30: // 		udiIDXOFFS_MaxPos		: UDINT := 16#0000_000E;	// 8B
	fbADSWRITE.WRITE			:= TRUE;
	fbADSWRITE.IDXOFFS			:= 16#0000_000E;
	fbADSWRITE.LEN				:= 8;
	fbADSWRITE.SRCADDR			:= ADR(lrSetMaxPos);
	iStepWrite					:= iStepWrite + 5;
		
35: // 	End
	fbADSWRITE.WRITE			:= FALSE;
	IF NOT fbADSWRITE.BUSY AND NOT fbADSWRITE.ERR THEN
		bBusy 					:= FALSE;
		iStepWrite				:= 0;
	ELSIF fbADSWRITE.ERR THEN
		iStepWrite				:= 1000;
	END_IF
	
1000:
	bBusy 						:= FALSE;
	bError 						:= TRUE;
	udiErrorID					:= fbADSWRITE.ERRID;
	iStepWrite					:= 0;

END_CASE
END_ACTION

END_FUNCTION_BLOCK

// ---- POUs/NC/FB_CalculateSpeed.TcPOU
(********************************************************************************)
(*							Beckhoff Automation Poland							*)
(*							FB_CalculateSpeed  v1.0								*)
(*									28.8.2013									*)
(*			Blok funkcyjny obliczający predkosc z pozycji. z filtracją wyjscia	*)
(*						Wewnatrz wykorzystany blok FB_Filter					*)
(*______________________________________________________________________________*)
FUNCTION_BLOCK FB_CalculateSpeed
VAR_INPUT
	dwInput					: DWORD;     			(* zliczone impulsy z enkodera *)
	tSamplingTime 			: TIME;     			(* czas cyklu odczytu wejscia dwInput, musi byc rowony lub wiekszy od cyklu programu *)
	tT						: TIME;					(* stala czasowa filtracji - po tym czasie wyjscie przyjmuje ok 0,65 wartosci wejsciowej*)
END_VAR
VAR_OUTPUT
	rOut					: REAL; 				(* aktualna prędkość - unit/ms*)
	bError					: BOOL;					(* blad - czas probkowania mniejszy niz czas cyklu *)
END_VAR

VAR
	dwPrevInput				: DWORD;		 		(*liczba impulsów z poprzedniego odczytu*)
	rSamplingTime			: REAL; 				(*czas cyklu odczytu wejscia dwInput *)
	rDistance				: REAL;   				(*roznica w odczycie pomiedzy probkowaniami*)
	rRawOut					: REAL;   				(*prędkość przed filtracją*)
	dwBound					: DWORD;				(*granica wyznaczajaca przepetlenie*)
	BIndex					: BYTE;					(* nr tasku - do porowniania czasu cyklu *)
	tCycleTime				: TIME;					(* Ustawiony czas Tasku w ms*)
	tCurrentTime			: TIME;					(* aktualny czas *)
	tLastTime				: TIME;					(* poprzedni czas *)
	bCalculate				: BOOL;					(* sygnal do wykonania obliczen *)
	fbFilter 				: FB_Filter;			(* blok filtracji *)
	fbGETCURTASKINDEX		: GETCURTASKINDEX; 		(* Blok sprawdzajcy numer Tasku *)
END_VAR
VAR CONSTANT
	dwMaxInput				: DWORD := 4294967295;	(*maksymalna liczba impulsów*)
END_VAR

fbGETCURTASKINDEX(index=> BIndex);

dwBound 		:= dwMaxInput/4;								(*graniczna wartosc roznicy impulsow jest rowna 25% maksymalnej wartosci*)
tCycleTime		:= UDINT_TO_TIME(_TaskInfo[BIndex].CycleTime/10000);
bError			:= tSamplingTime < tCycleTime;					(* sprawdzenie warunku wykonalnosci *)
rSamplingTime	:= TIME_TO_REAL(tSamplingTime);
tCurrentTime 	:= TIME();										(* pobranie czasu plc *)
bCalculate 		:= (tCurrentTime - tLastTime) >= tSamplingTime; 	(* sprawdzamy czy nadszedl czas obliczen *)

IF bCalculate AND NOT bError  THEN
	IF dwInput < dwBound AND dwPrevInput > dwMaxInput- dwBound THEN 		(* Przepetlenie na + *)
		rDistance := DWORD_TO_REAL(dwInput - dwPrevInput);
	ELSIF dwInput > dwMaxInput- dwBound AND dwPrevInput < dwBound THEN 	(* Przepetlenie na - *)
		rDistance := DWORD_TO_REAL(dwInput - dwPrevInput);
	ELSE																		(* Bez przepetlenia zwykle odejmowanie *)
		rDistance := DWORD_TO_REAL(dwInput - dwPrevInput);
	END_IF
	rRawOut := rDistance/rSamplingTime;										(* Obliczenie predkosci *)
	(* Przepisanie starych wartosci *)
	tLastTime 		:= tCurrentTime;
	dwPrevInput 	:= dwInput;
END_IF

(*wygladzanie przebiegu*)
fbFIlter(In := rRawOut, tSamplingTime:= tSamplingTime, tMeasureTime:= tT, Out => rOut);

END_FUNCTION_BLOCK

// ---- POUs/Various/FB_Filter.TcPOU
(****************************************************************************************)
(*							Beckhoff Automation Poland									*)
(*								FB_Filter  v1											*)
(*									27.05.2008											*)
(*				Bloczek do filtru inercyjnego do wygladzania przebiegow					*)
(* 			Uwaga!! w nowych aplikacjach nalezy stosowac FB_FilterEx 					*)
(*______________________________________________________________________________________*)
FUNCTION_BLOCK FB_Filter
VAR_INPUT
	In:						REAL;(*sygnal wejsciowy*)
	tSamplingTime:			TIME;(*czas probkowania*)
	tMeasureTime:			TIME;(*stala czasowa*)
END_VAR
VAR_OUTPUT
	Out:					REAL;(*sygnal wyjsciowy*)
END_VAR
VAR
	czas_probkowania_real:	REAL;
	stala_czasowa_real:		REAL;
	CLOCK: 					TP;
	lastOut: 				REAL;
	lastStan: 				BOOL;
	stan: 					BOOL;
END_VAR

CLOCK();
clock.PT:=tSamplingTime;
czas_probkowania_real:=TIME_TO_REAL(tSamplingTime);
stala_czasowa_real:= TIME_TO_REAL(tMeasureTime);
IF CLOCK.Q=FALSE THEN
	CLOCK(IN:=FALSE);
	stan := NOT stan;
	CLOCK(IN:=TRUE);
END_IF
IF(lastStan <> stan) THEN
	Out:= lastOut + (In -lastOut)*czas_probkowania_real/stala_czasowa_real;
END_IF
lastOut:=Out;
lastStan:= stan;

END_FUNCTION_BLOCK

// ---- POUs/NC/FB_Enc20bitToDWORD.TcPOU
(********************************************************************************************)
(*							Beckhoff Automation Poland										*)
(*								FB_Enc20bitToDWORD  v2										*)
(*									20.07.2010												*)
(*	Blok funkcyjny do poszerzania zakresu odczytu z encoderow,								*)
(*	wartosc wejsciowa typu DWORD przystosowana do 20 bitow <0; 1048575>						*)
(*	przenoszona jest na wyjscie typu DWORD <0; 4294967295>									*)
(*	Przepetlenie wartosci wejsciowej nie powoduje w tym przypadku bledu						*)
(*__________________________________________________________________________________________*)
FUNCTION_BLOCK FB_Enc20bitToDWORD
VAR_INPUT
	dwInput: 		DWORD;					(* wartosc wejsciowa *)
END_VAR
VAR_IN_OUT
	dwOutput: 		DWORD;					(*wartosc wyjsciowa*)
END_VAR
VAR
	dwLastInput: 	DWORD;
	mask20: 		DWORD := 16#000FFFFF;	(*20 bitow, 1048575 Dec*)
	dwOutputHW:		DWORD; 					(*Gorna czesc dworda*)
	bFirstCycle:	BOOL := TRUE;
END_VAR
VAR CONSTANT
	dwLow: 			DWORD := 250000;
	dwHigh: 		DWORD := 800000;
END_VAR

dwInput := mask20 AND dwInput;

(*pierwszy cykl*)
IF bFirstCycle THEN
	dwOutputHW := dwOutput AND 16#FFF00000;
	bFirstCycle := FALSE;
ELSE
	IF dwInput < dwLow AND dwLastInput > dwHigh THEN
		(*Przekroczylismy zakres w gore*)
		dwOutputHW := dwOutputHW + 16#00100000;
	END_IF

	IF dwInput > dwHigh AND dwLastInput < dwLow THEN
		(*Przekroczylismy zakres w dol*)
		dwOutputHW := dwOutputHW - 16#00100000;
	END_IF
END_IF

dwLastInput := dwInput;
dwOutput := dwOutputHW + dwInput;

END_FUNCTION_BLOCK

// ---- POUs/NC/FB_EncIntToDint.TcPOU
(****************************************************************************************)
(*							Beckhoff Automation Poland									*)
(*								FB_EncIntToDint  v1.1									*)
(*									2.12.2010											*)
(*	Blok funkcyjny do poszerzania zakresu odczytu z encoderow,							*)
(*	wartosc wejsciowa typu UINT <-32768; 32767>											*)
(*	przenoszona jest na wyjscie typu UDINT <-2147483648; 2147483647>					*)
(*	Przepetlenie wartosci wejsciowej nie powoduje w tym przypadku bledu					*)
(*______________________________________________________________________________________*)
FUNCTION_BLOCK FB_EncIntToDint
VAR_INPUT
	iInput : 			INT; 		(* wartosc wejsciowa *)
	bReset : 			BOOL;
END_VAR
VAR
	iDelta: 			INT;
	iLastInput : 		INT;
END_VAR
VAR_IN_OUT
	diOutput: 			DINT;		(* wartosc wyjsciowa  - warto zrobic jako persistent*)
END_VAR

IF bReset THEN
	diOutput := 0;
ELSE
	iDelta := ( iInput - iLastInput);
	diOutput := diOutput + iDelta;
END_IF

iLastInput := iInput;

END_FUNCTION_BLOCK

// ---- POUs/NC/FB_EncWordtoDword.TcPOU
(****************************************************************************************************)
(*							Beckhoff Automation Poland												*)
(*								FB_EncWordToDword  v1.1												*)
(*									2.12.2010														*)
(*	Blok funkcyjny do poszerzania zakresu odczytu z encoderow,										*)
(*	wartosc wejsciowa typu WORD <0;  65535> przenoszona jest na wyjscie typu DWORD <0; 4294967295>	*)
(*	Przepetlenie wartosci wejsciowej nie powoduje w tym przypadku bledu								*)
(*__________________________________________________________________________________________________*)
FUNCTION_BLOCK FB_EncWordToDword
VAR_INPUT
	wInput: 		DWORD;		(* wartosc wejsciowa *)
	bReset: 		BOOL; 		(* reset wartosci *)
END_VAR
VAR_IN_OUT
	dwOutput: 		DWORD;		(*wartosc wyjsciowa - warto zrobic jako presistent *)
END_VAR
VAR
	wLastInput: 	DWORD;		(* Ostatnia wartosc *)
	dwOutputHW:		DWORD; 		(* Gorna czesc dworda*)
	bFirstCycle: 	BOOL := TRUE;
END_VAR
VAR CONSTANT
	wLow: 			DWORD := 15000;
	wHigh:			DWORD := 50000;
END_VAR

(*pierwszy cykl*)
IF bReset THEN
	dwOutput := 0;
	dwOutputHW := 0;
END_IF

IF bFirstCycle THEN
	dwOutputHW := dwOutput AND 16#FFFF0000; (* pobranie gornego worda *)
	bFirstCycle := FALSE;
ELSE
	IF wInput < wLow AND wLastInput > wHigh THEN
		(* Przekroczylismy zakres w gore *)
		dwOutputHW := dwOutputHW + 16#00010000;
	END_IF
	IF wInput > wHigh AND wLastInput < wLow THEN
		(*Przekroczylismy zakres w dol*)
		dwOutputHW := dwOutputHW - 16#00010000;
	END_IF
END_IF

wLastInput := wInput;
dwOutput := dwOutputHW + wInput;

END_FUNCTION_BLOCK

// ---- POUs/NC/FB_ForceLockUnlock.TcPOU
(************************************************************************************************)
(*							Beckhoff Automation Poland											*)
(*								FB_ForceLockUnlock  v1.0										*)
(*									2.12.2010													*)
(*	Blok funkcyjny pozwalający w prosty sposób włączać i wyłączac hamulec silnika AMxxxx 		*)
(*							Potrzebna biblioteka MC2Drive 										*)
(*______________________________________________________________________________________________*)
FUNCTION_BLOCK FB_ForceLockUnlock
VAR_INPUT
	bForceLock : 		BOOL;
	bForceUnlock: 		BOOL;
END_VAR
VAR_OUTPUT
	bError: 			BOOL;
	bUnlocked: 			BOOL;
END_VAR
VAR_IN_OUT
	Axis: 				AXIS_REF;
END_VAR
VAR
	wWriteData:			WORD; 				(*1 - lock, 2 - unlock *)
	wReadData: 			WORD;
	ftWrite: 			F_TRIG;
	Delay1: 			TOF;
	fbSoEWrite: 		FB_SoEWrite;
	fbSoERead: 			FB_SoERead;
	wWriteDataOld: 		WORD;
END_VAR

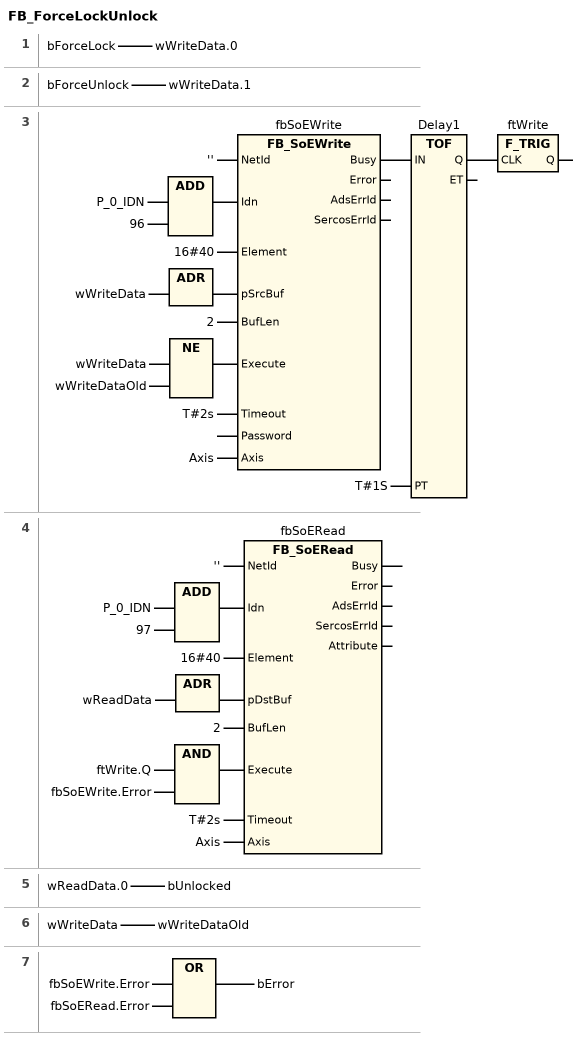
// NETWORK 1
wWriteData.0 := bForceLock;

// NETWORK 2
wWriteData.1 := bForceUnlock;

// NETWORK 3
fbSoEWrite(
    NetId := '',
    Idn := P_0_IDN + 96,
    Element := 16#40,
    pSrcBuf := ADR(wWriteData),
    BufLen := 2,
    Execute := wWriteData <> wWriteDataOld,
    Timeout := T#2s,
    Axis := Axis); // FB_SoEWrite
Delay1(IN := fbSoEWrite.Busy, PT := T#1S); // TOF
ftWrite(CLK := Delay1.Q); // F_TRIG

// NETWORK 4
fbSoERead(
    NetId := '',
    Idn := P_0_IDN + 97,
    Element := 16#40,
    pDstBuf := ADR(wReadData),
    BufLen := 2,
    Execute := ftWrite.Q AND fbSoEWrite.Error,
    Timeout := T#2s,
    Axis := Axis); // FB_SoERead

// NETWORK 5
bUnlocked := wReadData.0;

// NETWORK 6
wWriteDataOld := wWriteData;

// NETWORK 7
bError := fbSoEWrite.Error OR fbSoERead.Error;

END_FUNCTION_BLOCK

// ---- POUs/NC/FB_I2T_AX2000.TcPOU
(****************************************************************************)
(*							Beckhoff Automation Poland						*)
(*								FB_I2T_AX2000	 v1.0						*)
(*									27.05.2014								*)
(*							Blok odczytujący parametr I2T					*)
(* 							Wymaga biblioteki TcMc2Drive.lib 				*)
(*__________________________________________________________________________*)
FUNCTION_BLOCK FB_I2T_AX2000
VAR_INPUT
	bEnable					: BOOL := TRUE;
	sNetId					: T_AmsNetId; (* AMS Net ID of EtherCAT Master *)
	nSlaveAddr				: INT;
END_VAR
VAR_OUTPUT
	rI2T					: REAL;
	bBusy					: BOOL;
	bError					: BOOL;
	nErrId					: UDINT;
END_VAR
VAR
	fbEcCoESdoRead			: FB_EcCoESdoRead;
	tonWait200ms			: TON;
	dwI2T					: DWORD;
END_VAR

tonWait200ms(IN:= NOT tonWait200ms.Q AND bEnable, PT:=T#200MS );

fbEcCoESdoRead(
	sNetId:=sNetId ,
	nSlaveAddr:=INT_TO_UINT(nSlaveAddr),
	nSubIndex:=16#1 ,
	nIndex:=16#3559 ,
	pDstBuf:=ADR(dwI2T) ,
	cbBufLen:=SIZEOF(dwI2T) ,
	bExecute:=tonWait200ms.Q ,
	tTimeout:=t#2000ms ,
	bBusy=>bBusy ,
	bError=>bError ,
	nErrId=>nErrId );

rI2T := (DWORD_TO_REAL (dwI2T))/10.0;

END_FUNCTION_BLOCK

// ---- POUs/NC/FB_I2T_EL72x1.TcPOU
(************************************************************************************************)
(*							Beckhoff Automation Poland											*)
(*								FB_I2T_EL72x1	 v1.2											*)
(*							v1.1 - usuniecie /10, zmiana wyjść na typ USINT						*)
(*							v1.2 - poprawiony blad w nazwie zmiennej							*)
(*									24.10.2014													*)
(*							Blok odczytujący parametr I2T										*)
(* 							Wymaga biblioteki TcEtherCAT.lib 									*)
(*______________________________________________________________________________________________*)
FUNCTION_BLOCK FB_I2T_EL72x1
VAR_INPUT
(* A010:11 Amplifier I2T temperature  I2T model load Unit: % UINT8*)
(* A011:11 Motor I2T temperature  I2T model load Unit: % UINT8*)
	bEnable					: BOOL := TRUE; 		(* Pozwolenie na odczyt *)
	sNetId					: T_AmsNetId; 			(* AMS Net ID of EtherCAT Master *)
	nSlaveAddr				: UINT; 				(* Numer EtherCAT Slave *)
END_VAR
VAR_OUTPUT
	bBusy					: BOOL;
	bError					: BOOL;
	nErrorID				: UDINT;
	usiAmplifier_I2T		: USINT;
	usiMotor_I2T			: USINT;
END_VAR
VAR
(* Energy store/delete *)
	fbEcCoeSdoRead			: FB_EcCoESdoRead;
	bA010					: BOOL	:=TRUE;
	ftRead					: F_TRIG;
	tonWait200ms			: TON;
END_VAR

tonWait200ms(IN:=NOT tonWait200ms.Q AND bEnable, PT:=T#200MS );

fbEcCoeSdoRead.nIndex := SEL(bA010, 16#A011, 16#A010);
fbEcCoeSdoRead.pDstBuf := SEL(bA010, ADR(usiMotor_I2T), ADR(usiAmplifier_I2T));

fbEcCoeSdoRead(
	sNetId:= sNetId,
	nSlaveAddr:= nSlaveAddr,
	nSubIndex:= 16#11,
	cbBufLen:= 1,
	bExecute:= bEnable AND tonWait200ms.Q,
	bBusy=> bBusy,
	bError=> bError,
	nErrId=> nErrorID);

ftRead(CLK:= bBusy, Q=> );
bA010 := SEL(ftRead.Q, bA010, NOT bA010);

END_FUNCTION_BLOCK

// ---- POUs/NC/FB_PWM_BASIC.TcPOU
(********************************************************************************************************)
(*								Beckhoff Automation Poland												*)
(* 									FB_PWM_BASIC v1.1													*)
(* 										22.04.2010														*)
(*	v 1.1 - dodano bEnable, rCycleTime, początkowa faza to wyjście załączone, końcowa wyłączone			*)
(* 		Blok funkcyjny sterowania wyjsciem bOut typu BOOL na zasadzie modulowania szerokosci impulsu.	*)
(*					 Dokladnosc szerokosci impulsu  do 1 cylku sterownika.								*)
(* 							Konieczne jest dodanie biblioteki TcSystem									*)
(*______________________________________________________________________________________________________*)
FUNCTION_BLOCK FB_PWM_BASIC
VAR_INPUT
	bEnable: 			BOOL	:=TRUE;	(* Pozwolenie na działanie bloczka *)
	tPulseWidth: 		TIME; 			(*Szerokosc impulsu = 100% w ms typ zmiennej TIME*)
	fUpPercent: 		REAL; 			(*Aktualne procentowe wypelnienie impulsu*)
	rCycleTime: 		REAL;			(* Czas cylku - task, w milisekundach *)
END_VAR
VAR_OUTPUT
	bOut: 				BOOL;			(* Wyjscie *)
	wOn: 				WORD;			(* Liczba cykli z załączonym wyjściem *)
	wOff: 				WORD;			(* Liczba cykli z wyłaczonym wyjściem *)
END_VAR
VAR
	fCyclePulseWidth: 	REAL;  			(*Dlugosc impulsu = 100% w cyklach typ zmiennej REAL *)
	fCyclesOn: 			REAL;			(*Ilosc cykli, w ktorych sygnal jest zalaczony*)
	State: 				BYTE:=1;		(*Zmienna wyboru w instrukcji CASE*)
	(*Przeliczenie na pelne cykle*)
	wWidth: 			WORD;
	wCycleCounter:		WORD;			(*Licznik cykli zalaczenia/wylaczenia*)
	(*Przechowanie wartosci do porownania*)
	tPulseWidthOld: 	TIME	:= T#0MS;
	fUpPercentOld: 		REAL	:= -1;
END_VAR

IF bEnable THEN
	(*Przelicz tylko gdy zmienia sie dane*)
	IF tPulseWidth <> tPulseWidthOld OR fUpPercent <> fUpPercentOld THEN
		(*Sprawdzamy poprawnosc wprowadzonych danych*)
		IF fUpPercent <0 THEN fUpPercent := 0; END_IF
		IF fUpPercent > 100 THEN fUpPercent := 100; END_IF
		(*Obliczamy*)
		fCyclePulseWidth := TIME_TO_REAL(tPulseWidth)/rCycleTime; (*Dlugosc impulsu*)
		fCyclesOn := fCyclePulseWidth * fUpPercent/100;(*Cykle zalaczenia*)
	
		(*Przeliczamy na pelne cykle*)
		(*Opcja dla dokladniejszego przyblizenia impulsu On i Off*)
		wWidth := REAL_TO_WORD(fCyclePulseWidth);
		wOn := REAL_TO_WORD(fCyclesOn);
		(* Jeśli nie ma takiej potrzeby, nie wystawiaj wyjscia *)
		IF wOff = 0 THEN State := 0; END_IF
		wOff := REAL_TO_WORD(fCyclePulseWidth - fCyclesOn);
		(*Podstawiamy*)
		tPulseWidthOld := tPulseWidth;
		fUpPercentOld := fUpPercent;
	END_IF

	(*Albo wystawiamy TRUE albo FALSE*)
	CASE State OF
		0:
			bOut := FALSE;									(*Ustaw bOut na FALSE*)
			wCycleCounter := wCycleCounter  +  1;			(*Dodaj cykl do licznika*)
			IF wCycleCounter >= wOff THEN					(*Jezeli bylo bOut = FALSE wystarczajaca ilosc cykli to...*)
				wCycleCounter := 0;							(*Resetuj licznik*)
				IF wOff <> wWidth THEN State := 1; END_IF 	(*Przelacz tylko jesli ma byc kiedys bOut = TRUE*)
			END_IF
		1:
			bOut := TRUE;									(*Ustaw bOut na TRUE*)
			wCycleCounter := wCycleCounter  +  1;			(*Dodaj cykl do licznika*)
			IF wCycleCounter >= wOn THEN					(*Jezeli bylo bOut = TRUE wystarczajaca ilosc cykli to...*)
				wCycleCounter := 0;							(*Resetuj licznik*)
				IF wOn <> wWidth THEN State := 0; END_IF 	(*Przelacz tylko jesli ma byc kiedys bOut = FALSE*)
			END_IF
	END_CASE
ELSE
	bOut := FALSE;
	wCycleCounter := 0;
	State := 1;
END_IF

END_FUNCTION_BLOCK

// ---- POUs/NC/FB_SetBiasValue.TcPOU
(************************************************************************************************)
(*							Beckhoff Automation Poland											*)
(*								FB_SetBiasValue	 v1.0											*)
(*									12.04.2015													*)
(*							Blok wpisujący offset pozycji										*)
(* 							Wymaga biblioteki TcMc2.lib 										*)
(*______________________________________________________________________________________________*)
FUNCTION_BLOCK FB_SetBiasValue
VAR_INPUT
	bExecute			: BOOL; 		(* Narastajace zbocze aktywuje zapis *)
	sNetId				: T_AmsNetId;
	lrBias				: LREAL;
END_VAR
VAR_OUTPUT
	bBusy				: BOOL;
	bError				: BOOL;
	udiErrorID			: UDINT;
END_VAR
VAR_IN_OUT
	Axis				: AXIS_REF;
END_VAR
VAR
	fbADSWRITE			: ADSWRITE;
END_VAR

fbADSWRITE(
	NETID:= sNetId,
	PORT:= AMSPORT_R0_NC,
	IDXGRP:= 16#5000+Axis.NcToPlc.AxisId,
	IDXOFFS:= 7,
	LEN:= SIZEOF(lrBias),
	SRCADDR:= ADR(lrBias),
	WRITE:= bExecute,
	TMOUT:= ,
	BUSY=> bBusy,
	ERR=> bError,
	ERRID=> udiErrorID);

END_FUNCTION_BLOCK

// ---- POUs/NC/FB_TorqueMonitoringEL_Ex2.TcPOU
(****************************************************************************************************)
(*							Beckhoff Automation Poland												*)
(*							FB_TorqueMonitoringEL_Ex2 v1.1											*)
(*									25.11.2015														*)
(*																									*)
(*	Blok funkcyjny pozwala na monitorowanie i ograniczanie momentu oraz monitoring parametru I2T	*)
(*									dla EL7211.														*)
(*	Zmienne do zlinkowania zadeklarowane są wewnątrz bloku.		 									*)
(*	Ograniczenie i monitorowanie momentu															*)
(*	Ograniczenie momentu podawane jest przez wejście rTorqueLimit. 									*)
(*	Na wyjściu podana jest wartość surowa w %, jak i przeskalowana na A (prąd) i Nm (moment). 		*)
(*	Blok zwraca wartości bieżące, przefiltrowane i maksymalne. 										*)
(*	Wartości maksymalne mogą być wyzerowane za pomocą zmiennej bReset. 								*)
(*	Wewnętrznie wykorzystany jest blok FB_Filter.													*)
(*		I2T: 	Określamy okno czasowe pomiaru														*)
(* 	Wymaga biblioteki TcMc2Drive.lib 																*)
(*__________________________________________________________________________________________________*)
FUNCTION_BLOCK FB_TorqueMonitoringEL_Ex2
	VAR_INPUT
	bCalculate					: BOOL		:= TRUE;				(* Calculation request - initial value - TRUE *)
	bReset						: BOOL 		:= TRUE; 				(* Calculation request - initial value - TRUE *)
	rTorqueLimit				: REAL 		:= 100.0;			 	(* 0.0-100.0 %, rozdzielczość 0.1% *)
	tI2T_Window					: TIME;
END_VAR
VAR_OUTPUT
	bError						: BOOL; 							(* Communication error *)
	iErrorID					: INT;
	iTorque 			AT %I*	: INT; 								(* Raw data *)
	rCurrent					: REAL;								(* [A] *)
	rTorque						: REAL;								(* [Nm] *)
	rCurrentF					: REAL;								(* Filtered *)
	rTorqueF					: REAL;								(* Filtered *)
	rCurrentMax					: REAL;								(* Max *)
	rTorqueMax					: REAL;								(* Max *)
	rI2T						: REAL 		:= 0.0;
	rI2TMax						: REAL 		:= 0.0;
END_VAR
VAR_IN_OUT
	Axis						: AXIS_REF;
END_VAR
VAR
	iStep						: INT 		:= 0;

	rtCalculate					: R_TRIG;
	iTorqueLimitValue  	AT %Q*	:INT; 								(* Raw dara*)
	rFactor						: REAL;								(* iTorque -1000..1000 --> - rPeakCurrent .. rPeakCurrent *)
	rTorqueConstant				: REAL; 							(* [Nm/A] *)
	rPeakCurrent				: REAL; 							(* [A] *)
	rRatedCurrent				: REAL; 							(* [A] *)

	fbFilter					: FB_Filter;

	sNetId						: T_AmsNetId;
	uiSlaveAddr					: UINT;

	rI2T_pom					: REAL 		:= 0.0;
	rI2T_Window					: REAL;
	bFlag_1						: BOOL		:= FALSE;
	iCycles						: INT;
	rCycleTime_pom     	        : REAL;
	iCounter					: INT;
	rBuffer						: ARRAY[1..100] OF REAL;
	rBuffer_2					: ARRAY[1..100] OF REAL;

	fbMC_ReadDriveAddress		: MC_ReadDriveAddress;

	rCycleTime      		    : REAL;                             (* Ustawiony czas Tasku w ms*)
	fbGETCURTASKINDEX   		: GETCURTASKINDEX;                 	(* Blok sprawdzajcy numer Tasku *)
	BIndex                      : BYTE;                             (* Nr Tasku *)
(*-----------------------------------------------------------------------------------------------------------------------*)
	bRead						: BOOL;
	tTime						: TIME;
	wInfo						: WORD;
	dwPeakCurrent				: DWORD;
	dwStadnstillCurrent			: DWORD;
	dwRatedCurrent				: DWORD;
	dwTorqueConstant			: DWORD;
	dwDClinkCV					: DWORD		:= 0;
	fbEcCoESdoRead				: FB_EcCoESdoRead;
	BSubIndex					: BYTE;
	wIndex						: WORD;
	i							: INT		:= 1;
	pDstBuf						: POINTER TO DWORD;
	cbBufLen					: UDINT;
	ftRead						: F_TRIG;
	tonRead						: TON;
END_VAR

rtCalculate(CLK:= bCalculate, Q=> );
IF rtCalculate.Q THEN
	iStep := 0;
END_IF

CASE iStep OF

0:

(*Read drive adress*)

	bError:=FALSE;
	iErrorID:=0;
	fbMC_ReadDriveAddress(Execute := TRUE,Axis := Axis);
	iStep := iStep + 10;
10:
	fbMC_ReadDriveAddress(Axis := Axis);
	IF fbMC_ReadDriveAddress.Done THEN
		fbMC_ReadDriveAddress.Execute := FALSE;
		sNetId := fbMC_ReadDriveAddress.DriveAddress.NetID;
		uiSlaveAddr := fbMC_ReadDriveAddress.DriveAddress.SlaveAddress;
		iStep := iStep + 10;
	ELSIF fbMC_ReadDriveAddress.Error THEN
		iStep:=999;
		iErrorID:=UDINT_TO_INT(fbMC_ReadDriveAddress.ErrorID);
	END_IF
20:

(*Read cycle time*)

	fbGETCURTASKINDEX(index => BIndex);
	rCycleTime := UDINT_TO_REAL(_TaskInfo[BIndex].cycleTime)/10000.0;

(*Calculate algorithm sampling time*)

	rI2T_Window := TIME_TO_REAL(tI2T_Window);
	rCycleTime_pom := rI2T_Window/100 ;
	IF rCycleTime_pom < rCycleTime THEN
		rCycleTime_pom := rCycleTime;
	END_IF
	tTime := REAL_TO_TIME(rCycleTime_pom);
	iStep := iStep + 10;
30:

(*Chceck motor information using CoE*)

	bRead := TRUE;
	iStep := iStep + 10;
40:
	CoE_Read();
	IF NOT bRead THEN
		iStep := iStep + 10;
	END_IF
50:

(*Calculate current and torque value*)

	rCurrent := INT_TO_REAL(iTorque)*rPeakCurrent/1000;
	rTorque := rCurrent * rTorqueConstant;

(*Filter curent value*)

	fbFilter(In:= rCurrent, tSamplingTime:= REAL_TO_TIME(rCycleTime), tMeasureTime:= REAL_TO_TIME(rCycleTime_pom), Out=> rCurrentF);
	rTorqueF := rCurrentF * rTorqueConstant;

(*Save torque and current max values*)

	IF rCurrentMax < rCurrentF THEN
		rCurrentMax := rCurrentF;
		rTorqueMax := rTorqueF;
	END_IF

(*b_Flag_1 is set to TRUE when PLC cycle matches with algorythm sampling rate*)

	IF rCycleTime <> 0 THEN
		IF iCycles < rCycleTime_pom/rCycleTime  THEN
			iCycles := iCycles + 1;
			bFlag_1 := FALSE;
		ELSE
			iCycles := 0;
			bFlag_1 := TRUE;
		END_IF
	END_IF

(*Save momentary I2T values in ring buffer*)

	IF bFlag_1 THEN
		FOR iCounter:=1 TO 99 DO
			rBuffer[iCounter] := rBuffer[iCounter+1];
			rBuffer_2[iCounter] := rBuffer_2[iCounter+1];
		END_FOR
		rBuffer[100] := rCurrentF *rCurrentF* rCycleTime_pom;
		rBuffer_2[100] := rRatedCurrent *rRatedCurrent* rCycleTime_pom;
	END_IF
	rI2T := 0;
	rI2T_pom := 0;

(*Calculate I2T parameter*)

	FOR iCounter:=1 TO 100 DO
		rI2T := rI2T + rBuffer[iCounter];
		rI2T_pom := rI2T_pom + rBuffer_2[iCounter];
	END_FOR

(*Scale I2T to 0-100% range*)

	IF rI2T_pom <> 0  THEN
		rI2T := rI2T/rI2T_pom*100;
	END_IF

	IF rI2TMax < rI2T THEN
		rI2TMax := rI2T;
	END_IF

	IF bReset THEN
		rCurrentMax := 0;
		rTorqueMax := 0;
		rI2TMax := 0;
		FOR iCounter:=1 TO 100 DO
			rBuffer[iCounter] := 0;
			rBuffer_2[iCounter] := 0;
		END_FOR;
	END_IF
999:

(* Error occured *)

	bError:=TRUE;
	fbMC_ReadDriveAddress(Execute := FALSE,Axis := Axis);
	fbEcCoESdoRead(
	sNetId:= sNetId,
	nSlaveAddr:= uiSlaveAddr,
	nSubIndex:= BSubIndex,
	nIndex:= wIndex,
	pDstBuf:= pDstBuf,
	cbBufLen:= cbBufLen,
	bExecute := FALSE);

END_CASE;
iTorqueLimitValue := REAL_TO_INT(LIMIT(0.0,(rTorqueLimit)*10,1000.0));

ACTION CoE_Read:
CASE i OF
1:
	wIndex 			:= 16#6010;
	BSubIndex 		:= 1;
	pDstBuf 		:= ADR (wInfo);
	cbBufLen 		:= SIZEOF(wInfo);
2:
	wIndex 			:= 16#8011;
	BSubIndex 		:= 16#11;
	pDstBuf 		:= ADR (dwPeakCurrent);
	cbBufLen 		:= SIZEOF(dwPeakCurrent);
3:
	wIndex 			:= 16#8011;
	BSubIndex 		:= 16#12;
	pDstBuf 		:= ADR (dwRatedCurrent);
	cbBufLen 		:= SIZEOF(dwRatedCurrent);
4:
	wIndex 			:= 16#8011;
	BSubIndex 		:= 16#16;
	pDstBuf 			:= ADR (dwTorqueConstant);
	cbBufLen 		:= SIZEOF(dwTorqueConstant);
ELSE
	bRead 			:= FALSE;

	rRatedCurrent		:= DWORD_TO_REAL(dwRatedCurrent)/1000;
	rPeakCurrent 		:= DWORD_TO_REAL(dwPeakCurrent)/1000.0;
	rTorqueConstant	:= DWORD_TO_REAL(dwTorqueConstant)/1000.0;

	i := 1;
END_CASE

tonRead(IN := NOT tonRead.Q AND bRead, PT:= tTime, Q=> , ET=> );

fbEcCoESdoRead(
	sNetId:= sNetId,
	nSlaveAddr:= uiSlaveAddr,
	nSubIndex:= BSubIndex,
	nIndex:= wIndex,
	pDstBuf:= pDstBuf,
	cbBufLen:= cbBufLen,
	bExecute := tonRead.Q);
ftRead(CLK:= fbEcCoESdoRead.bBusy, Q=> );
IF ftRead.Q THEN
	IF fbEcCoESdoRead.bError THEN
		iErrorID := UDINT_TO_INT(fbEcCoESdoRead.nErrId);
		iStep:=999;
	END_IF
	i := i+1;
END_IF
END_ACTION

END_FUNCTION_BLOCK

// ---- POUs/NC/FB_TorqueMonitoringEx2.TcPOU
(****************************************************************************************************)
(*							Beckhoff Automation Poland												*)
(*							FB_TorqueMonitoringEx2 v1.1												*)
(*									23.04.2015														*)
(*			v1.1 - poprawiona obsługa błedów, optymalizacja obliczeń								*)
(*	Blok funkcyjny pozwala na monitorowanie i ograniczanie momentu oraz monitoring parametru I2T	*)
(*									dla AX5xxx.														*)
(*	Zmienne do zlinkowania zadeklarowane są wewnątrz bloku. 										*)
(*					Ograniczenie i monitorowanie momentu											*)
(*	Ograniczenie momentu podawane jest przez wejście rTorqueLimit. 									*)
(*	Na wyjściu podana jest wartość surowa w %, jak i przeskalowana na A (prąd) i Nm (moment).	 	*)
(*	Blok zwraca wartości bieżące, przefiltrowane i maksymalne. 										*)
(*	Wartości maksymalne mogą być wyzerowane za pomocą zmiennej bReset. 								*)
(*	Wewnętrznie wykorzystany jest blok FB_Filter.													*)
(*		I2T: 	Określamy okno czasowe pomiaru														*)
(* 	Wymaga biblioteki TcMc2Drive.lib 																*)
(*__________________________________________________________________________________________________*)
FUNCTION_BLOCK FB_TorqueMonitoringEx2
VAR_INPUT
	bCalculate					: BOOL		 := TRUE; 				(* Calculation request - initial value - TRUE *)
	bReset						: BOOL		 := TRUE;				(* Calculation request - initial value - TRUE *)
	rTorqueLimit				: REAL		 := 100.0; 				(* 0.0-100.0 %, rozdzielczość 0.1% *)
	tI2T_Window					: TIME		 :=T#1M;
END_VAR
VAR_OUTPUT
	bError						: BOOL; 							(* Communication error *)
	uiErrorID					: UINT;
	iTorque 			AT %I*	: INT; 								(* Raw data, linked to Torque feedback value AT, S-0-0084 *)
	rCurrent					: REAL; 							(* [A] *)
	rTorque						: REAL; 							(* [Nm] *)
	rCurrentF					: REAL;								(* Filtered *)
	rTorqueF					: REAL;								(* Filtered *)
	rCurrentMax					: REAL;								(* Max *)
	rTorqueMax					: REAL;								(* Max *)
	rI2T						: REAL; 							(* % nominal *)
	rI2TMax						: REAL;
END_VAR
VAR_IN_OUT
	Axis						: AXIS_REF;
END_VAR
VAR
	rtCalculate					: R_TRIG;
	fbSoERead					: FB_SoERead;
	iStep						: INT;
	P_0_0092_Value				: DWORD;
	P_0_0093_Value				: DWORD;
	P_0_0070_Value				: WORD;
	S_0_0111_Value				: DWORD;
	iBipolarTorqueLimitValue  	AT %Q*:		INT; 					(* Raw data, linked to Bipolar torque limit value MDT, S-0-0092 *)
	rPeakCurrent				: REAL; 							(* P_0_0092_Value in [A] *)
	rFactor						: REAL; 							(* iTorque -1000..1000 --> - rPeakCurrent .. rPeakCurrent *)
	rContinuousStallTorque		: REAL;								(* P_0_0070_Value [Nm] *)
	rContinuousStallCurrent		: REAL;								(* S_0_0111_Value [A] *)
	rTorqueConstant				: REAL; 							(* P_0_0070_Value/S_0_0111_Value [Nm/A] *)
	fbFilter					: FB_Filter;

	rI2T_pom					: REAL 		:= 0.0;
	rRatedCurrent				: REAL;	 							(* P_0_0093_Value in [A] *)
	rI2T_Window					: REAL;
	bFlag_1						: BOOL 		:= FALSE;
	bFlag_2						: BOOL 		:= FALSE;
	iCycles						: INT;
	iCycles_pom					: INT;
	rCycleTime_pom				: REAL;
	iCounter					: INT;
	rBuffer						: ARRAY[1..100] OF REAL;
	rBuffer_2					: ARRAY[1..100] OF REAL;

	rCycleTime					: REAL;                            	(* Ustawiony czas Tasku w ms*)
	fbGETCURTASKINDEX   		: GETCURTASKINDEX;                 	(* Blok sprawdzajcy numer Tasku *)
	BIndex						: BYTE;                             (* Nr Tasku *)
END_VAR

rtCalculate(CLK:= bCalculate, Q=> );
IF rtCalculate.Q THEN iStep := 0; END_IF

CASE iStep OF
	0: (*Init*)
	bError := FALSE;
	iStep := iStep+ 10;

	10: (*Read P_0_0092*)
	fbSoERead.Idn 		:= P_0_IDN + 92;
	fbSoERead.Element	:= EC_SOE_ELEMENT_VALUE;
	fbSoERead.pDstBuf	:= ADR(P_0_0092_Value);
	fbSoERead.BufLen	:= SIZEOF(P_0_0092_Value);
	fbSoERead.Execute	:= TRUE;
	iStep := iStep+ 5;

	15:
	IF NOT fbSoERead.Busy AND NOT fbSoERead.Error THEN
		rPeakCurrent := DWORD_TO_REAL(P_0_0092_Value)/1000.0;
		rFactor := DWORD_TO_REAL(P_0_0092_Value)/1000000.0;
		fbSoERead.Execute	:= FALSE;
		iStep := iStep+ 5;
	END_IF
	IF fbSoERead.Error THEN
		iStep := 100;
	END_IF

	20:
	(*Read P_0_0070*)
	fbSoERead.Idn 		:= P_0_IDN + 70;
	fbSoERead.Element	:= EC_SOE_ELEMENT_VALUE;
	fbSoERead.pDstBuf	:= ADR(P_0_0070_Value);
	fbSoERead.BufLen	:= SIZEOF(P_0_0070_Value);
	fbSoERead.Execute	:= TRUE;
	iStep := iStep+ 5;

	25:
	IF NOT fbSoERead.Busy AND NOT fbSoERead.Error THEN
		rContinuousStallTorque := WORD_TO_REAL(P_0_0070_Value)/100;
		fbSoERead.Execute	:= FALSE;
		iStep := iStep+ 5;
	END_IF
	IF fbSoERead.Error THEN
		iStep := 100;
	END_IF

	30: (* Read S_0_0111*)
	fbSoERead.Idn 		:= S_0_IDN + 111;
	fbSoERead.Element	:= EC_SOE_ELEMENT_VALUE;
	fbSoERead.pDstBuf	:= ADR(S_0_0111_Value);
	fbSoERead.BufLen	:= SIZEOF(S_0_0111_Value);
	fbSoERead.Execute	:= TRUE;
	iStep := iStep+ 5;

	35:
	IF NOT fbSoERead.Busy AND NOT fbSoERead.Error THEN
		rContinuousStallCurrent := DWORD_TO_REAL(S_0_0111_Value)/1000;
		rTorqueConstant := rContinuousStallTorque/rContinuousStallCurrent;
		fbSoERead.Execute	:= FALSE;
		iStep := iStep+ 5;
	END_IF
	IF fbSoERead.Error THEN
		iStep := 100;
	END_IF

	40: (* Read P_0_0093*)
	fbSoERead.Idn 		:= P_0_IDN + 93;
	fbSoERead.Element	:= EC_SOE_ELEMENT_VALUE;
	fbSoERead.pDstBuf	:= ADR(P_0_0093_Value);
	fbSoERead.BufLen	:= SIZEOF(P_0_0093_Value);
	fbSoERead.Execute	:= TRUE;
	iStep := iStep+ 5;

	45:
	IF NOT fbSoERead.Busy AND NOT fbSoERead.Error THEN
		rRatedCurrent := DWORD_TO_REAL(P_0_0093_Value)/1000;
		fbSoERead.Execute	:= FALSE;
		iStep := iStep+ 5;
	END_IF
	IF fbSoERead.Error THEN
		iStep := 100;
	END_IF

	50: (*Calculations*)
	rCurrent := INT_TO_REAL(iTorque) * rFactor;
	rTorque := rCurrent * rTorqueConstant;

	100:
	iStep := 0;
	fbSoERead(Execute:= FALSE,Axis:= Axis);
	bError := TRUE;
	uiErrorID := fbSoERead.AdsErrId;
END_CASE

(*Read cycle time*)
fbGETCURTASKINDEX(index => BIndex);
rCycleTime := UDINT_TO_REAL(_TaskInfo[BIndex].cycleTime)/10000.0;

(*Calculate algorithm sampling time*)
rI2T_Window := TIME_TO_REAL(tI2T_Window);
rCycleTime_pom := rI2T_Window/100 ;

IF rCycleTime_pom < rCycleTime THEN
	rCycleTime_pom := rCycleTime;
END_IF

(*Filter current value*)

fbFilter(In:= rCurrent, tSamplingTime:= REAL_TO_TIME(rCycleTime), tMeasureTime:= REAL_TO_TIME(rCycleTime_pom), Out=> rCurrentF);
rTorqueF := rCurrentF * rTorqueConstant;

(*Save torque and current max values*)
IF rCurrentMax < rCurrentF THEN
	rCurrentMax := rCurrentF;
	rTorqueMax := rTorqueF;
END_IF

(*b_Flag_1 is set to TRUE when PLC cycle matches with algorythm sampling rate*)

IF rCycleTime <> 0 THEN
	IF iCycles < rCycleTime_pom/rCycleTime  THEN
		iCycles := iCycles + 1;
		bFlag_1 := FALSE;
	ELSE
		iCycles := 0;
		bFlag_1 := TRUE;
	END_IF
END_IF

(*Save momentary I2T values in ring buffer*)

IF bFlag_1 THEN
	FOR iCounter :=1 TO 99 DO
		rBuffer[iCounter] := rBuffer[iCounter+1];
		rBuffer_2[iCounter] := rBuffer_2[iCounter+1];
	END_FOR
	rBuffer[100] := rCurrentF *rCurrentF* rCycleTime_pom;
	rBuffer_2[100] := rRatedCurrent *rRatedCurrent* rCycleTime_pom;
END_IF

rI2T := 0;
rI2T_pom := 0;

(*Calculate I2T parameter*)

FOR iCounter:=1 TO 100 BY 1 DO
	rI2T := rI2T + rBuffer[iCounter];
	rI2T_pom := rI2T_pom + rBuffer_2[iCounter];
END_FOR

(*Scale I2T to 0-100% range*)

IF rI2T_pom  <> 0  THEN
	rI2T := rI2T/rI2T_pom*100;
END_IF

IF rI2TMax < rI2T THEN
	rI2TMax := rI2T;
END_IF

IF bReset THEN
	rCurrentMax := 0;
	rTorqueMax := 0;
	rI2TMax := 0;
	FOR iCounter:=1 TO 100 BY 1 DO
		rBuffer[iCounter] := 0;
		rBuffer_2[iCounter] := 0;
	END_FOR;
END_IF
iBipolarTorqueLimitValue := REAL_TO_INT(LIMIT(0.0,(rTorqueLimit)*10,1000.0));

fbSoERead(
	NetId:= '',
	Timeout:= T#1s,
	Axis:= Axis);

END_FUNCTION_BLOCK

// ---- POUs/Switches/FB_2SwB.TcPOU
(****************************************************************************************)
(*							Beckhoff Automation Poland									*)
(*								FB_2SwB v1.1											*)
(*									9.11.2007											*)
(*				Blok funkcyjny symulujący pracę dwóch przycisków bistabilnych			*)
(*						 jako sterowania światłem schodowym								*)
(*______________________________________________________________________________________*)
FUNCTION_BLOCK FB_2SwB
VAR_INPUT
	bSwitch1:			BOOL;		(*Pierwszy przycisk bistabilny*)
	bSwitch2:			BOOL;		(*Drugi przycisk bistabilny*)
	bReset:				BOOL;		(*Przywrócenie stanu początkowego*)
END_VAR
VAR_OUTPUT
	bOut:				BOOL;		(*Wyjscie sterujące oświetleniem*)
END_VAR
VAR
	RTrig1:				R_TRIG;
	RTrig2:				R_TRIG;
	FTrig1:				F_TRIG;
	FTrig2:				F_TRIG;
END_VAR

RTrig1(CLK:= bSwitch1);
RTrig2(CLK:= bSwitch2);
FTrig1(CLK:= bSwitch1);
FTrig2(CLK:= bSwitch2);
bOut  := SEL(RTrig1.Q OR rTrig2.Q OR FTrig1.Q OR FTrig2.Q, bOut , NOT bOut );
IF bReset THEN bOut := FALSE; END_IF

END_FUNCTION_BLOCK

// ---- POUs/Switches/FB_2SwM.TcPOU
(****************************************************************************************)
(*							Beckhoff Automation Poland									*)
(*								FB_2SwM v1.1											*)
(*									9.11.2007											*)
(*				Blok funkcyjny symulujący pracę dwóch przycisków monostabilnych			*)
(*						 jako sterowania światłem schodowym								*)
(*______________________________________________________________________________________*)
FUNCTION_BLOCK FB_2SwM
VAR_INPUT
	bSwitch1:	BOOL;		(*Pierwszy przycisk monostabilny*)
	bSwitch2:	BOOL;		(*Drugi przycisk monostabilny*)
	bReset:		BOOL; 		(*Przywrócenie stanu początkowego*)
END_VAR
VAR_OUTPUT
	bOut:		BOOL; 		(*Wyjscie sterujące oświetleniem*)
END_VAR
VAR
	Trig1:		R_TRIG;
	Trig2:		R_TRIG;
END_VAR

Trig1(CLK:= bSwitch1);
Trig2(CLK:= bSwitch2);
bOut  := SEL(Trig1.Q OR Trig2.Q, bOut , NOT bOut );
IF bReset THEN bOut := FALSE; END_IF

END_FUNCTION_BLOCK

// ---- POUs/Switches/FB_Click.TcPOU
(********************************************************************************************************)
(*							Beckhoff Automation Poland													*)
(*								FB_Click	 v1.1														*)
(*								16.06.2008																*)
(*	Blok funkcyjny rozpoznajacy pojedyncze klikniecie, klikniecie podwojne lub nacisniecie przycisku	*)
(*______________________________________________________________________________________________________*)
FUNCTION_BLOCK FB_Click
VAR_INPUT
	bSwitch: 		BOOL;		 		(*Przycisk*)
	tTime: 			TIME 	:= T#1S; 	(*Czas kiedu mozna kliknac dwukrotnie*)
	tPress: 		TIME := T#500MS;	(*Rozpoznanie nacisniecia*)
END_VAR
VAR_OUTPUT
	bDouble: 		BOOL;(*Przyjmuje wartosc TRUE dla dwukrotnego klikniecia*)
	bSingle: 		BOOL;(*Przyjmuje wartosc TRUE dla pojedynczego klikniecia*)
	bPress: 		BOOL;(*Przyjmuje wartosc TRUE dla przytrzymania przycisku*)
END_VAR
VAR
	nCounter: 		SINT;
	timer: 			TON;
	timerPress: 	TON;
	rtrig: 			R_TRIG;
	ftrig: 			F_TRIG;
	pom: 			BOOL; 				(*zmienna pomocnicza*)
END_VAR

(*Zeby tylko przez jeden cykl byly ustawione wyjscia*)
bDouble := FALSE;
bSingle := FALSE;

timer(IN:= , PT:=tTime , Q=> , ET=> );
timerPress(IN:= bSwitch, PT:= tPress, Q=>bPress , ET=> );
rtrig(CLK:= bSwitch, Q=> );
ftrig(CLK:= bSwitch, Q=> );

(*Wyzerowanie licznika jak jest Press*)
IF timerPress.Q THEN
	nCounter := 0;
END_IF

(*Obsługa krótkiego sygnału*)
IF rtrig.Q THEN
	timer.IN := TRUE;
	pom := TRUE;
END_IF
IF ftrig.Q AND pom THEN
	pom := FALSE;
	nCounter := nCounter + 1;
END_IF

IF timer.Q THEN
	timer.IN := FALSE;
	IF nCounter = 1 THEN
		bSingle := TRUE;
	ELSIF nCounter > 1 THEN
		bDouble := TRUE;
	END_IF
	nCounter := 0;
END_IF

END_FUNCTION_BLOCK

// ---- POUs/Switches/FB_ClickCounterBit.TcPOU
(********************************************************************************************************)
(*							Beckhoff Automation Poland													*)
(*							FB_ClickCounterBit v1.0														*)
(*									18.02.2008															*)
(*				Blok funkcyjny zliczający ilość kliknięć i podający ją w formie bitu w bajcie			*)
(*______________________________________________________________________________________________________*)
FUNCTION_BLOCK FB_ClickCounterBit
VAR_INPUT
	bSwitch:		BOOL;(*Przycisk, którego kliknięcia zliczamy*)
	tInterval: 		TIME;(*max czas między kliknięciami*)
END_VAR
VAR_OUTPUT
	BOut:			BYTE;(*Zliczona ilość kliknięć*)
END_VAR
VAR
	Counting:		TOF;
	BAmount:		BYTE;
	RisingEdge:		R_TRIG;
	FallingEdge:	F_TRIG;
END_VAR

Counting(IN:=bSwitch , PT:= tInterval, Q=> , ET=> );
RisingEdge(CLK:= bSwitch, Q=> );
FallingEdge(CLK:= Counting.Q, Q=> );
IF RisingEdge.Q AND Counting.Q THEN
	BAmount := BAmount+1;
	BOut := 0;
END_IF
IF FallingEdge.Q THEN
	IF BAmount > 8 THEN
		BAmount := 8;
	END_IF(**)
	BOut := LREAL_TO_BYTE(EXPT(2,BAmount-1));
	BAmount := 0;
END_IF

END_FUNCTION_BLOCK

// ---- POUs/Switches/FB_ClickCounterByte.TcPOU
(********************************************************************************************)
(*							Beckhoff Automation Poland										*)
(*							FB_ClickCounterByte v1.0										*)
(*									18.02.2008												*)
(*				Blok funkcyjny zliczający ilość kliknięć i podający ją w formie bajtu		*)
(*__________________________________________________________________________________________*)
FUNCTION_BLOCK FB_ClickCounterByte
VAR_INPUT
	bSwitch:		BOOL;		(*Przycisk, którego kliknięcia zliczamy*)
	tInterval: 		TIME;		(*max czas między kliknięciami*)
END_VAR
VAR_OUTPUT
	BOut:			BYTE;		(*Zliczona ilość kliknięć*)
END_VAR
VAR
	Counting:		TOF;
	BAmount:		BYTE;
	RisingEdge:		R_TRIG;
	FallingEdge:	F_TRIG;
END_VAR

Counting(IN:=bSwitch , PT:= tInterval, Q=> , ET=> );
RisingEdge(CLK:= bSwitch, Q=> );
FallingEdge(CLK:= Counting.Q, Q=> );
IF RisingEdge.Q AND Counting.Q THEN
	BAmount := BAmount+1;
END_IF
IF FallingEdge.Q THEN
	BOut := BAmount;
	BAmount := 0;
ELSE
	BOut := 0;
END_IF

END_FUNCTION_BLOCK

// ---- POUs/Switches/FB_Dimmer1P.TcPOU
(****************************************************************************************)
(*							Beckhoff Automation Poland									*)
(*								FB_Dimmer1P v1.0										*)
(*									21.11.2007											*)
(*		Blok funkcyjny do przyciemniania/rozjaśniania za pomocą 1 przycisku bistabilnego*)
(*							wykorzystywany z KL2751										*)
(*______________________________________________________________________________________*)
FUNCTION_BLOCK FB_Dimmer1P
VAR_INPUT
	bSwitch:		BOOL;					(*Obsługiwany przycisk*)
	bReset:			BOOL; 					(*Reset bloku funkcyjnego przez funkcję centralną*)
END_VAR
VAR_OUTPUT
	iOut: 			INT;					(*Wyjscie - powinno byc zlinkowane z wyjściem modułu KL2751*)
END_VAR
VAR_IN_OUT
	iOldOut: 		INT;					(*Zapamiętanie stanu w yjścia*)
END_VAR
VAR
	tLong:			TIME	:=T#200MS;		(*Czas określający długie wciśnięcie przycisku*)
	iStep:			INT		:=100;			(*Krok zmany wyjścia*)
	Czas:			TON;
	Licznik:		CTU;
	iFunction:		INT;
	bLong: 			BOOL	:=TRUE;
	bShort: 		BOOL;
	ResetTrig:		R_TRIG;
END_VAR

(*Przywrócenie ustawień początkowych*)
ResetTrig(CLK:=bReset);
IF ResetTrig.Q THEN iFunction := 1; bLong := TRUE; bShort := FALSE;  END_IF;

(* Wykrycie dlugiego nacisniecia *)
Czas(IN:= bSwitch, PT:=tLong);
(* Rozpoznanie funkcji *)
Licznik(CU:= bSwitch, RESET:= Licznik.Q, PV:= 2);

IF Licznik.CV = 0 AND bSwitch THEN iFunction := 0; END_IF;(*wlaczany przycisk, byc moze rozjasnianie*)
IF Licznik.CV = 0 AND NOT bSwitch THEN iFunction := 1; END_IF;(*wylaczony przycisk, byc moze wlaczenie*)
IF Licznik.CV = 1 AND bSwitch THEN iFunction := 2; END_IF;(*wlaczany przycisk, byc moze sciemnianie*)
IF Licznik.CV = 1 AND NOT bSwitch THEN iFunction := 3; END_IF;(*wylaczony przycisk, byc moze wylaczenie*)
(*zapamietanie, ze bylo krotkie nacisniecie*)
IF bSwitch AND NOT Czas.Q THEN bLong := FALSE; END_IF;
IF NOT bSwitch AND NOT bLong THEN bShort := TRUE; END_IF;
(*zapamietanie, ze bylo dlugie nacisniecie*)
IF bSwitch AND Czas.Q THEN bLong := TRUE; bShort := FALSE; END_IF;

CASE iFunction OF

0:
(*przyciemnianie*)
IF bLong THEN
	iOut:=iOut-iStep;
	IF iOut<iStep THEN
		iOut :=0;
	END_IF
	iOldOut:=iOut;
END_IF;

1:
(*wylaczenie*)
IF bShort THEN iOut := 0; END_IF;

2:
(*rozjasnianie*)
IF bLong THEN
	iOut:=iOut+iStep;
	IF iOut<0THEN
		iOut :=32767;
	END_IF
	iOldOut:=iOut;
END_IF;

3:
(*wlaczenie*)
IF bShort THEN iOut:=iOldOut; END_IF;

END_CASE;

END_FUNCTION_BLOCK

// ---- POUs/Switches/FB_Dimmer1PMinMax.TcPOU
(****************************************************************************************)
(*							Beckhoff Automation Poland									*)
(*							FB_Dimmer1PMinMax v1.0										*)
(*									21.11.2007											*)
(*		Blok funkcyjny do przyciemniania/rozjaśniania za pomocą 1 przycisku bistabilnego*)
(*					z określaniem poziomu minimalnego i maksymalnego oświetlenia		*)
(*							wykorzystywany z KL2751										*)
(*______________________________________________________________________________________*)
FUNCTION_BLOCK FB_Dimmer1PMinMax
VAR_INPUT
	bSwitch:		BOOL;			(*Obsługiwany przycisk*)
	iMinLevel: 		INT; 			(*Minimalna wartość wyjścia*)
	iMaxLevel:	 	INT; 			(*Maksymalna wartość wyjścia*)
	bReset:			BOOL; 			(*Reset bloku funkcyjnego przez funkcję centralną*)
END_VAR
VAR_OUTPUT
	iOut: 			INT;			(*Wyjscie - powinno byc zlinkowane z wyjściem modułu KL2751*)
END_VAR
VAR_IN_OUT
	iOldOut: 		INT;			(*Zapamiętanie stanu w yjścia*)
END_VAR
VAR
	tLong:			TIME:=T#200MS;	(*Czas określający długie wciśnięcie przycisku*)
	iStep:			INT:=100;		(*Krok zmany wyjścia*)
	Czas:			TON;
	Licznik:		CTU;
	iFunction:		INT;
	bLong: 			BOOL:=TRUE;
	bShort: 		BOOL;
	ResetTrig:		R_TRIG;
END_VAR

(*Przywrócenie ustawień początkowych*)
ResetTrig(CLK:=bReset);
IF ResetTrig.Q THEN iFunction := 1; bLong := TRUE; bShort := FALSE;  END_IF;

(* Wykrycie dlugiego nacisniecia *)
Czas(IN:= bSwitch, PT:=tLong);
(* Rozpoznanie funkcji *)
Licznik(CU:= bSwitch, RESET:= Licznik.Q, PV:= 2);

IF Licznik.CV = 0 AND bSwitch THEN iFunction := 0; END_IF;(*wlaczany przycisk, byc moze rozjasnianie*)
IF Licznik.CV = 0 AND NOT bSwitch THEN iFunction := 1; END_IF;(*wylaczony przycisk, byc moze wlaczenie*)
IF Licznik.CV = 1 AND bSwitch THEN iFunction := 2; END_IF;(*wlaczany przycisk, byc moze sciemnianie*)
IF Licznik.CV = 1 AND NOT bSwitch THEN iFunction := 3; END_IF;(*wylaczony przycisk, byc moze wylaczenie*)
(*zapamietanie, ze bylo krotkie nacisniecie*)
IF bSwitch AND NOT Czas.Q THEN bLong := FALSE; END_IF;
IF NOT bSwitch AND NOT bLong THEN bShort := TRUE; END_IF;
(*zapamietanie, ze bylo dlugie nacisniecie*)
IF bSwitch AND Czas.Q THEN bLong := TRUE; bShort := FALSE; END_IF;

CASE iFunction OF

0:
(*przyciemnianie*)
IF bLong THEN
	iOut:=iOut-iStep;
	IF iOut<iMinLevel+iStep THEN
		iOut :=iMinLevel;
	END_IF
	iOldOut:=iOut;
END_IF;

1:
(*wylaczenie*)
IF bShort THEN iOut := 0; END_IF;

2:
(*rozjasnianie*)
IF bLong THEN
	iOut:=iOut+iStep;
	IF iOut<0 OR iOut>iMaxLevel THEN
		iOut :=iMaxLevel;
	END_IF
	iOldOut:=iOut;
END_IF;

3:
(*wlaczenie*)
IF bShort THEN iOut:=iOldOut; END_IF;

END_CASE;

END_FUNCTION_BLOCK

// ---- POUs/Switches/FB_Dimmer2P.TcPOU
(********************************************************************************************)
(*							Beckhoff Automation Poland										*)
(*								FB_Dimmer2P v1.0											*)
(*									21.11.2007												*)
(*		Blok funkcyjny do przyciemniania/rozjaśniania za pomocą 1 przycisków bistabilnych	*)
(*							wykorzystywany z KL2751											*)
(*__________________________________________________________________________________________*)
FUNCTION_BLOCK FB_Dimmer2P
VAR_INPUT
	bSwitchOnUp:			BOOL;			(*Przycisk 1*)
	bSwitchOffDown:			BOOL;			(*Przycisk 2*)
	bReset:					BOOL;			(*Reset bloku funkcyjnego przez funkcję centralną*)
END_VAR
VAR_OUTPUT
	iOut: 					INT;			(*Wyjscie - powinno byc zlinkowane z wyjściem modułu KL2751*)
END_VAR
VAR_IN_OUT
	iOldOut: 				INT;			(*Zapamiętanie stanu w yjścia*)
END_VAR
VAR
	iStep:					INT:=100;		(*Krok zmany wyjścia*)
	timeLong:		 		TIME:=T#200MS;	(*Czas długiego kliknięcia*)
	ftrig1:					F_TRIG;
	ftrig2:					F_TRIG;
	rtrig1:					R_TRIG;
	rtrig2:					R_TRIG;
	timer1:					TON;
	timer2:					TON;
	pom1: 					BOOL;
	bLong1: 				BOOL;
	bLong2: 				BOOL;
	pom2: 					BOOL;
	ResetTrig: 				R_TRIG;
END_VAR

(*Przywrócenie ustawień początkowych*)
ResetTrig(CLK:=bReset);
IF ResetTrig.Q THEN
	iOut :=0;
END_IF;
(*Wywołanie trigerow i timerow*)
timer1(PT:= timeLong);
ftrig1(CLK:= bSwitchOnUp);
rtrig1(CLK:= bSwitchOnUp);
timer2(PT:= timeLong);
ftrig2(CLK:= bSwitchOffDown);
rtrig2(CLK:= bSwitchOffDown);
(*Przycisk On i Up*)
(*Włączenie przycisku*)
IF rtrig1.Q THEN
	timer1.IN := TRUE;
	pom1 := TRUE;
	bLong1 := FALSE;
END_IF
(*Krótkie wciśnięcie*)
IF ftrig1.Q AND pom1 THEN
	pom1 := FALSE;
	timer1.IN := FALSE;
	iOut := iOldOut;
	bLong1 := FALSE;
END_IF
(*Długie wciśnięcie*)
IF timer1.Q THEN
	timer1.IN := FALSE;
	bLong1 := TRUE;
	pom1 := FALSE;
END_IF
(*Operacje gdy długi Up*)
IF bLong1 THEN
	iOut:=iOut+iStep;
	IF iOut<0THEN
		iOut :=32767;
	END_IF
	iOldOut:=iOut;
END_IF;
(*Wyłączenie długiego wciśnięcia*)
IF NOT bSwitchOnUp THEN
	bLong1 := FALSE;
END_IF

(*Przycisk Off i Down*)
(*Włączenie przycisku*)
IF rtrig2.Q THEN
	timer2.IN := TRUE;
	pom2 := TRUE;
	bLong2 := FALSE;
END_IF
(*Krótkie wciśnięcie*)
IF ftrig2.Q AND pom2 THEN
	pom2 := FALSE;
	timer2.IN := FALSE;
	iOut := 0;
	bLong2 := FALSE;
END_IF
(*Długie wciśnięcie*)
IF timer2.Q THEN
	timer2.IN := FALSE;
	bLong2 := TRUE;
	pom2 := FALSE;
END_IF
(*Operacje gdy długi Off*)
IF bLong2 THEN
	iOut:=iOut-iStep;
	IF iOut<iStep THEN
		iOut :=0;
	END_IF
	iOldOut:=iOut;
END_IF;
(*Wyłączenie długiego wciśnięcia*)
IF NOT bSwitchOffDown THEN
	bLong2 := FALSE;
END_IF

END_FUNCTION_BLOCK

// ---- POUs/Switches/FB_Dimmer2PMinMax.TcPOU
(********************************************************************************************)
(*							Beckhoff Automation Poland										*)
(*							FB_Dimmer2PMinMax v1.0											*)
(*									21.11.2007												*)
(*		Blok funkcyjny do przyciemniania/rozjaśniania za pomocą 1 przycisków bistabilnych	*)
(*					z określaniem poziomu minimalnego i maksymalnego oświetlenia			*)
(*							wykorzystywany z KL2751											*)
(*__________________________________________________________________________________________*)
FUNCTION_BLOCK FB_Dimmer2PMinMax
VAR_INPUT
	bSwitchOnUp:			BOOL;				(*Przycisk 1*)
	bSwitchOffDown:			BOOL;				(*Przycisk 2*)
	iMinLevel: 				INT; 				(*Minimalna wartość wyjścia*)
	iMaxLevel:		 		INT; 				(*Maksymalna wartość wyjścia*)
	bReset:					BOOL; 				(*Reset bloku funkcyjnego przez funkcję centralną*)
END_VAR
VAR_OUTPUT
	iOut: 					INT;				(*Wyjscie - powinno byc zlinkowane z wyjściem modułu KL2751*)
END_VAR
VAR_IN_OUT
	iOldOut: 				INT;				(*Zapamiętanie stanu w yjścia*)
END_VAR
VAR
	iStep:					INT:=100;			(*Krok zmany wyjścia*)
	timeLong:		 		TIME:=T#200MS;		(*Czas długiego kliknięcia*)
	ftrig1:					F_TRIG;
	ftrig2:					F_TRIG;
	rtrig1:					R_TRIG;
	rtrig2:					R_TRIG;
	timer1:					TON;
	timer2:					TON;
	pom1: 					BOOL;
	bLong1: 				BOOL;
	bLong2: 				BOOL;
	pom2: 					BOOL;
	ResetTrig: 				R_TRIG;
END_VAR

(*Przywrócenie ustawień początkowych*)
ResetTrig(CLK:=bReset);
IF ResetTrig.Q THEN
	iOut :=0;
END_IF;
(*Wywołanie trigerow i timerow*)
timer1(PT:= timeLong);
ftrig1(CLK:= bSwitchOnUp);
rtrig1(CLK:= bSwitchOnUp);
timer2(PT:= timeLong);
ftrig2(CLK:= bSwitchOffDown);
rtrig2(CLK:= bSwitchOffDown);
(*Przycisk On i Up*)
(*Włączenie przycisku*)
IF rtrig1.Q THEN
	timer1.IN := TRUE;
	pom1 := TRUE;
	bLong1 := FALSE;
END_IF
(*Krótkie wciśnięcie*)
IF ftrig1.Q AND pom1 THEN
	pom1 := FALSE;
	timer1.IN := FALSE;
	iOut := iOldOut;
	bLong1 := FALSE;
END_IF
(*Długie wciśnięcie*)
IF timer1.Q THEN
	timer1.IN := FALSE;
	bLong1 := TRUE;
	pom1 := FALSE;
END_IF
(*Operacje gdy długi Up*)
IF bLong1 THEN
	iOut:=iOut+iStep;
	IF iOut<0 OR iOut>iMaxLevel THEN
		iOut :=iMaxLevel;
	END_IF
	iOldOut:=iOut;
END_IF;
(*Wyłączenie długiego wciśnięcia*)
IF NOT bSwitchOnUp THEN
	bLong1 := FALSE;
END_IF

(*Przycisk Off i Down*)
(*Włączenie przycisku*)
IF rtrig2.Q THEN
	timer2.IN := TRUE;
	pom2 := TRUE;
	bLong2 := FALSE;
END_IF
(*Krótkie wciśnięcie*)
IF ftrig2.Q AND pom2 THEN
	pom2 := FALSE;
	timer2.IN := FALSE;
	iOut := 0;
	bLong2 := FALSE;
END_IF
(*Długie wciśnięcie*)
IF timer2.Q THEN
	timer2.IN := FALSE;
	bLong2 := TRUE;
	pom2 := FALSE;
END_IF
(*Operacje gdy długi Off*)
IF bLong2 THEN
	iOut:=iOut-iStep;
	IF iOut<iMinLevel+iStep THEN
		iOut :=iMinLevel;
	END_IF
	iOldOut:=iOut;
END_IF;
(*Wyłączenie długiego wciśnięcia*)
IF NOT bSwitchOffDown THEN
	bLong2 := FALSE;
END_IF

END_FUNCTION_BLOCK

// ---- POUs/Switches/FB_ShortLong.TcPOU
(****************************************************************************************)
(*							Beckhoff Automation Poland									*)
(*								FB_ShortLong v2											*)
(*									2.04.2012											*)
(*	Bloczek do rozpoznania długiego/krotkiego wcisniecia przycisku						*)
(*______________________________________________________________________________________*)
FUNCTION_BLOCK FB_ShortLong
VAR_INPUT
	bSwitch: 			BOOL; 			(*Przycisk*)
	tLong: 				TIME;			(*Czas dlugiego wcisniecia*)
END_VAR
VAR_OUTPUT
	bShort: 			BOOL; 			(*TRUE gdy krotkie*)
	bLong: 				BOOL;			(*TRUE gdy dlugie*)
END_VAR
VAR
	t1: 				TON;
	ft1: 				F_TRIG;
END_VAR

ft1(CLK:= bSwitch , Q=> );
IF ft1.Q THEN
	bLong := t1.Q;
	bShort := NOT t1.Q;
END_IF
t1(IN:= bSwitch, PT:= tLong, Q=> , ET=> );

END_FUNCTION_BLOCK

// ---- POUs/Switches/FB_ShortLongTrig.TcPOU
(************************************************************************************)
(*							Beckhoff Automation Poland								*)
(*								FB_ShortLongTrig v2									*)
(*									2.04.2012										*)
(*	Bloczek do rozpoznania długiego/krotkiego wcisniecia przycisku- wyjscia			*)
(*__________________________________________________________________________________*)
FUNCTION_BLOCK FB_ShortLongTrig
VAR_INPUT
	bSwitch: 	BOOL; (*Przycisk*)
	tLong: 		TIME; (*Czas dlugiego wcisniecia*)
END_VAR
VAR_OUTPUT
	bShort: 	BOOL; (*TRUE gdy krotkie*)
	bLong: 		BOOL;(*TRUE gdy dlugie*)
END_VAR
VAR
	t1: 		TON;
	ft1: 		F_TRIG;
END_VAR

ft1(CLK:= bSwitch , Q=> );
IF ft1.Q THEN
	bLong := t1.Q;
	bShort := NOT t1.Q;
ELSE
	bLong := FALSE;
	bShort := FALSE;
END_IF
t1(IN:= bSwitch, PT:= tLong, Q=> , ET=> );

END_FUNCTION_BLOCK

// ---- POUs/Switches/FB_Sw4F.TcPOU
(********************************************************************************************)
(*							Beckhoff Automation Poland										*)
(*								FB_Sw4F v1.1												*)
(*									9.11.2007												*)
(*					Blok funkcyjny symulujący przycisk sterujący 4 wyjściami typu BOOL		*)
(*							bShortOn | bShortOff = TRUE | bLongOn | bLongOff				*)
(*__________________________________________________________________________________________*)
FUNCTION_BLOCK FB_Sw4F
VAR_INPUT
	bSwitch:			BOOL;					(*Obsługiwany przycisk*)
	tLong:				TIME	:=T#200MS;		(*Czas określający długie wciśnięcie przycisku*)
	bReset:				BOOL; 					(*Reset bloku funkcyjnego przez funkcję centralną*)
END_VAR
VAR_OUTPUT
	bShortOn:			BOOL;		 			(*Przyjmuje wartość TRUE dla krótkiego naciśnięcia podczas włączania*)
	bShortOff:			BOOL; 					(*Przyjmuje wartość TRUE dla krótkiego naciśnięcia podczas wyłączania*)
	bLongOn:			BOOL; 					(*Przyjmuje wartość TRUE dla długiego naciśnięcia podczas włączania*)
	bLongOff:			BOOL; 					(*Przyjmuje wartość TRUE dla długiego naciśnięcia podczas wyłączania*)
END_VAR
VAR
	iStep:				INT;
	Czas:				TON;
	Licznik:			CTU;
	bLong: 				BOOL	:=TRUE;
	bShort: 			BOOL;
	BOut:				BYTE; (*	xxxx 0001 - bShortOn
						xxxx 0010 - bShortOff
						xxxx 0100 - bLongOn
						xxxx 1000 - bLongOff
						*)
END_VAR

(*Przywrócenie ustawień początkowych*)
IF bReset THEN iStep := 1; bLong := TRUE; bShort := FALSE; BOut := 0; END_IF;

(* Wykrycie dlugiego nacisniecia *)
Czas(IN:= bSwitch, PT:=tLong);
(* Rozpoznanie funkcji *)
Licznik(CU:= bSwitch, RESET:= Licznik.Q, PV:= 2);

IF Licznik.CV = 0 AND bSwitch THEN iStep := 0; END_IF;(*wlaczany przycisk, byc moze rozjasnianie*)
IF Licznik.CV = 0 AND NOT bSwitch THEN iStep := 1; END_IF;(*wylaczony przycisk, byc moze wlaczenie*)
IF Licznik.CV = 1 AND bSwitch THEN iStep := 2; END_IF;(*wlaczany przycisk, byc moze sciemnianie*)
IF Licznik.CV = 1 AND NOT bSwitch THEN iStep := 3; END_IF;(*wylaczony przycisk, byc moze wylaczenie*)
(*zapamietanie, ze bylo krotkie nacisniecie*)
IF bSwitch AND NOT Czas.Q THEN bLong := FALSE; END_IF;
IF NOT bSwitch AND NOT bLong THEN bShort := TRUE; END_IF;
(*zapamietanie, ze bylo dlugie nacisniecie*)
IF bSwitch AND Czas.Q THEN bLong := TRUE; bShort := FALSE; END_IF;

CASE iStep OF

(*Wlaczenie i rozjasnianie*)
0:
(*dlugie nacisniecie >= tLong*)
IF bLong THEN BOut := 2#00001000; END_IF;

1:
(*Krotkie nacisniecie*)
IF bShort THEN BOut := 2#00000010; END_IF;

(*Przygaszanie i wylaczenie*)
2:
(*dlugie nacisniecie >= tLong*)
IF bLong THEN BOut := 2#00000100; END_IF;

3:
(*Krotkie nacisniecie*)
IF bShort THEN BOut := 2#00000001; END_IF;

END_CASE;

(*Wystawienie wyjść*)
	bShortOn := BOut.0;
	bShortOff := BOut.1;
	bLongOn := BOut.2;
	bLongOff := BOut.3;

END_FUNCTION_BLOCK

// ---- POUs/Switches/FB_Sw4FTrig.TcPOU
(********************************************************************************************)
(*							Beckhoff Automation Poland										*)
(*								FB_Sw4FTrig v1.1											*)
(*									9.11.2007												*)
(*					Blok funkcyjny symulujący przycisk sterujący 4 wyjściami typu BOOL		*)
(*							bShortOn | bShortOff = TRUE | bLongOn | bLongOff				*)
(*__________________________________________________________________________________________*)
FUNCTION_BLOCK FB_Sw4FTrig
VAR_INPUT
	bSwitch:		BOOL;					(*Obsługiwany przycisk*)
	tLong:			TIME	:=T#200MS;		(*Czas określający długie wciśnięcie przycisku*)
	bReset:			BOOL; 					(*Reset bloku funkcyjnego przez funkcję centralną*)
END_VAR
VAR_OUTPUT
	bShortOn:		BOOL; 					(*Przyjmuje wartość TRUE dla krótkiego naciśnięcia podczas włączania*)
	bShortOff:		BOOL; 					(*Przyjmuje wartość TRUE dla krótkiego naciśnięcia podczas wyłączania*)
	bLongOn:		BOOL; 					(*Przyjmuje wartość TRUE dla długiego naciśnięcia podczas włączania*)
	bLongOff:		BOOL; 					(*Przyjmuje wartość TRUE dla długiego naciśnięcia podczas wyłączania*)
END_VAR
VAR
	iStep:			INT;
	Czas:			TON;
	Licznik:		CTU;
	bLong: 			BOOL	:=TRUE;
	bShort: 		BOOL;
	BOut:			BYTE; (*	xxxx 0001 - bShortOn
						xxxx 0010 - bShortOff
						xxxx 0100 - bLongOn
						xxxx 1000 - bLongOff
						*)
	ResetTrig:		R_TRIG;
	ShortOnTrig:	R_TRIG;
	ShortOffTrig:	R_TRIG;
	LongOnTrig:		R_TRIG;
	LongOffTrig:	R_TRIG;
END_VAR

(*Przywrócenie ustawień początkowych*)
ResetTrig(CLK:=bReset);
IF ResetTrig.Q THEN iStep := 1; bLong := TRUE; bShort := FALSE; BOut := 0; END_IF;

(* Wykrycie dlugiego nacisniecia *)
Czas(IN:= bSwitch, PT:=tLong);
(* Rozpoznanie funkcji *)
Licznik(CU:= bSwitch, RESET:= Licznik.Q, PV:= 2);

IF Licznik.CV = 0 AND bSwitch THEN iStep := 0; END_IF;(*wlaczany przycisk, byc moze rozjasnianie*)
IF Licznik.CV = 0 AND NOT bSwitch THEN iStep := 1; END_IF;(*wylaczony przycisk, byc moze wlaczenie*)
IF Licznik.CV = 1 AND bSwitch THEN iStep := 2; END_IF;(*wlaczany przycisk, byc moze sciemnianie*)
IF Licznik.CV = 1 AND NOT bSwitch THEN iStep := 3; END_IF;(*wylaczony przycisk, byc moze wylaczenie*)
(*zapamietanie, ze bylo krotkie nacisniecie*)
IF bSwitch AND NOT Czas.Q THEN bLong := FALSE; END_IF;
IF NOT bSwitch AND NOT bLong THEN bShort := TRUE; END_IF;
(*zapamietanie, ze bylo dlugie nacisniecie*)
IF bSwitch AND Czas.Q THEN bLong := TRUE; bShort := FALSE; END_IF;

CASE iStep OF

(*Wlaczenie i rozjasnianie*)
0:
(*dlugie nacisniecie >= tLong*)
IF bLong THEN BOut := 2#00001000; END_IF;

1:
(*Krotkie nacisniecie*)
IF bShort THEN BOut := 2#00000010; END_IF;

(*Przygaszanie i wylaczenie*)
2:
(*dlugie nacisniecie >= tLong*)
IF bLong THEN BOut := 2#00000100; END_IF;

3:
(*Krotkie nacisniecie*)
IF bShort THEN BOut := 2#00000001; END_IF;

END_CASE;

(*Wystawienie wyjść*)
ShortOnTrig(CLK:= BOut.0, Q=>bShortOn );
ShortOffTrig(CLK:= BOut.1, Q=>bShortOff );
LongOnTrig(CLK:= BOut.2, Q=>bLongOn );
LongOffTrig(CLK:= BOut.3, Q=>bLongOff );

END_FUNCTION_BLOCK

// ---- POUs/Switches/FB_SwOrSen.TcPOU
(****************************************************************************************************)
(*							Beckhoff Automation Poland												*)
(*								FB_SwOrSen v1.1														*)
(*									9.11.2007														*)
(*	Blok funkcyjny symulujący przycisk bistabilny pracujacy w 3 trybach:							*)
(*	usMode = 0 - reaguje tylko na włącznik, nie reaguje na czujkę									*)
(*	usMode = 1 - reaguje tylko na czujkę, nie reaguje na włącznik									*)
(*	usMode = 2 - swiatło włączamy włącznikiem, a wyłącza sie przez czujkę							*)
(*	usMode = 3 - 	światło reaguje na czujkę,														*)
(*				jeżeli jednak włączono światło włącznikiem (nawet gdy było włączone prze czujnik),	*)
(*				to pomimo braku sygnału z czujnika, nie wyłączy się.								*)
(*__________________________________________________________________________________________________*)

FUNCTION_BLOCK FB_SwOrSen
VAR_INPUT
	bSwitch:			BOOL;				(*Włącznik światła*)
	bSensor:			BOOL;				(*Czujnik ruchu*)
	tDelay:				TIME;				(*Czas po jakim gaśnie światło podczas kontroli przez czujnik ruchu*)
	usMode:				USINT;				(*Wybór trybu pracy*)
END_VAR
VAR_OUTPUT
	bOut:				BOOL;				(*Wyjście sterujące oświetleniem*)
END_VAR
VAR
	Triger:				R_TRIG;
	Timer:				TOF;
	Timer_2:			TOF;
END_VAR

Triger();
Timer();
Timer_2();

IF usMode <> 0 AND usMode <> 1 AND usMode <>2 THEN usMode := 3; END_IF

CASE usMode OF

	0:
	(*swiatlo reaguje tylko na wlacznik*)
	bOut := bSwitch;

	1:
	(*swiatlo reaguje tylko na czujke*)
	Timer(IN:=NOT bSensor, PT:= tDelay );
	bOut := Timer.Q;

	2:
	(*swiatlo reaguje na czujke i wlacznik*)
	Triger(CLK:= bSwitch);
	Timer_2(IN:= Triger.Q, PT:= tDelay);
	Timer(IN:=NOT bSensor AND bSwitch, PT:= tDelay );
	bOut :=bSwitch AND (Timer.Q OR Timer_2.Q);

	3:
	Timer(IN:=NOT bSensor, PT:= tDelay );
	IF bSwitch THEN
	(*Przycisk włączony*)
		bOut := bSwitch;
	ELSE
	(*Przycisk wyłączony*)
		bOut := Timer.Q;
	END_IF

END_CASE

END_FUNCTION_BLOCK

// ---- POUs/Switches/FB_SwOrSenTrig.TcPOU
(****************************************************************************************************)
(*							Beckhoff Automation Poland												*)
(*								FB_SwOrSenTrig v1.1													*)
(*									9.11.2007														*)
(*	Blok funkcyjny symulujący przycisk monostabilny pracujacy w 3 trybach:							*)
(*	usMode = 0 - reaguje tylko na włącznik, nie reaguje na czujkę									*)
(*	usMode = 1 - reaguje tylko na czujkę, nie reaguje na włącznik									*)
(*	usMode = 2 - swiatło włączamy włącznikiem, a wyłącza sie przez czujkę							*)
(*	usMode = 3 - 	światło reaguje na czujkę,														*)
(*				jeżeli jednak włączono światło włącznikiem (nawet gdy było włączone prze czujnik),	*)
(*				to pomimo braku sygnału z czujnika, nie wyłączy się.								*)
(*__________________________________________________________________________________________________*)
FUNCTION_BLOCK FB_SwOrSenTrig
VAR_INPUT
	bSwitch:				BOOL;			(*Włącznik światła*)
	bSensor:				BOOL;			(*Czujnik ruchu*)
	tDelay:					TIME;			(*Czas po jakim gaśnie światło podczas kontroli przez czujnik ruchu*)
	usMode:					USINT;			(*Wybór trybu pracy*)
	bReset:					BOOL; 			(*Reset bloku funkcyjnego przez funkcję centralną*)
END_VAR
VAR_OUTPUT
	bOut:					BOOL;			(*Wyjście sterujące oświetleniem*)
END_VAR
VAR
	Triger:					R_TRIG;
	Timer:					TOF;
	Timer_2:				TOF;
	Stan_poprzedni:			BOOL;
END_VAR

Triger(CLK:= bSwitch);(*Wcisnięcie przycisku monostabilnego*)
Timer();
Timer_2();
IF bReset THEN bOut := FALSE; Stan_poprzedni := FALSE; END_IF
IF usMode <> 0 AND usMode <> 1 AND usMode <>2 THEN usMode := 3; END_IF

CASE usMode OF

	0:
	(*swiatlo reaguje tylko na wlacznik*)
	Stan_poprzedni := SEL(Triger.Q,Stan_poprzedni, NOT Stan_poprzedni);
	bOut := Stan_poprzedni;

	1:
	(*swiatlo reaguje tylko na czujke*)
	Timer(IN:=NOT bSensor, PT:= tDelay );
	bOut := Timer.Q;

	2:
	(*swiatlo reaguje na czujke i wlacznik*)
	Timer_2(IN:= NOT Stan_poprzedni AND  Triger.Q, PT:= tDelay);
	Stan_poprzedni := SEL(Triger.Q,Stan_poprzedni, NOT Stan_poprzedni);
	Timer(IN:=NOT bSensor AND Stan_poprzedni, PT:= tDelay );
	bOut := (Timer.Q AND Stan_poprzedni) OR Timer_2.Q;

	3:
	Stan_poprzedni := SEL(Triger.Q,Stan_poprzedni, NOT Stan_poprzedni);
	Timer(IN:=NOT bSensor, PT:= tDelay );
	IF Stan_poprzedni THEN
	(*Przycisk włączony*)
		bOut := Stan_poprzedni;
	ELSE
	(*Przycisk wyłączony*)
		bOut := Timer.Q;
	END_IF

END_CASE

END_FUNCTION_BLOCK

// ---- POUs/Various/FB_AnalogTo3Point.TcPOU
//==================================================================================================
//					Beckhoff Automation Poland
//							26.05.2017
//		Blok funkcyjny zmieniajacy wartosc ciagla w 3P
// 	v1.0 	|| TC v 3.1.4020.32 	|| - pierwsza wersja
//==================================================================================================
FUNCTION_BLOCK FB_AnalogTo3Point
VAR_INPUT
	bReset						: BOOL;
	rSetpoint					: REAL;
	tTaskCycleTime				: TIME;
	rMinSetpoint				: REAL;
	rMaxSetpoint				: REAL;
	rThreshold					: REAL;
	rTolerance					: REAL;
	tStrokeTime					: TIME := T#3M;
	tSwitchOverDeadTime			: TIME := T#5S;
END_VAR
VAR_OUTPUT
	bOpen						: BOOL;
	bClose						: BOOL;
	rPosition					: REAL;
	bError						: BOOL;
END_VAR
VAR
	rE							: REAL;		// Odchylka SP - CV
	rWholeDistance				: REAL;
	bMove						: BOOL;		// Flaga koniecznosci ruchu - ustawiana gdy odchylka jest wieksza niz rThreshold
	rStrokeTime					: REAL;
	rTaskCycleTime				: REAL;
	rSf							: REAL;
	rOneCycleDistance			: REAL;
	tofWaitOpen					: TOF;
	tofWaitClose				: TOF;
END_VAR

// Wywolanie FB
tofWaitOpen(IN:= bOpen, PT:= tSwitchOverDeadTime);
tofWaitClose(IN:= bClose, PT:= tSwitchOverDeadTime);
// Reset
IF bReset THEN
	tofWaitOpen(IN:= FALSE);
	tofWaitClose(IN:= FALSE);
	rPosition					:= rMinSetpoint;
	bOpen						:= FALSE;
	bClose						:= FALSE;
END_IF
// Sprawdzanie parametrów
bError							:= (rMinSetpoint >= rMaxSetpoint) 
								OR (rThreshold <= rTolerance)
								OR tTaskCycleTime = T#0MS
								OR tStrokeTime = T#0MS;
IF NOT bError THEN
	// Limit SP
	rSetpoint 					:= LIMIT(rMinSetpoint, rSetpoint, rMaxSetpoint);
	
	// Open/Close
	rE 							:= rSetpoint - rPosition;
	rWholeDistance				:= rMaxSetpoint - rMinSetpoint;
	bMove 						S= ABS(rE) > rThreshold;
	bMove 						R= ABS(rE) < rTolerance;
	bOpen						:= rE > 0 AND bMove AND NOT tofWaitClose.Q;//((rSetpoint - rPosition) >= rThreshold) AND bMove;// ;
	bClose						:= rE < 0 AND bMove AND NOT tofWaitOpen.Q;//((rPosition - rSetpoint) >= rThreshold) AND bMove;// ;
	
	// Position
	rTaskCycleTime 				:= TIME_TO_REAL(tTaskCycleTime);
	rStrokeTime 				:= TIME_TO_REAL(tStrokeTime);
	rSf							:= rTaskCycleTime/rStrokeTime;
	rOneCycleDistance			:= rSf * rWholeDistance;
	IF bOpen THEN
		rPosition 				:= rPosition + rOneCycleDistance;
	ELSIF bClose THEN
		rPosition 				:= rPosition - rOneCycleDistance;
	END_IF
	rPosition 					:= LIMIT(rMinSetpoint, rPosition, rMaxSetpoint);	
END_IF

END_FUNCTION_BLOCK

// ---- POUs/Various/FB_Average.TcPOU
(********************************************************************************************)
(*							Beckhoff Automation Poland										*)
(*								FB_Average	 v1.2											*)
(*									2.02.2011												*)
(*								v1.2 Optymalizacja wewnętrzna								*)
(*					Blok funkcyjny obliczający średnią z wartości wejściowej rValue			*)
(*					w zadanym przedziale czasowym lub z określonej ilości pomiarów			*)
(*__________________________________________________________________________________________*)
FUNCTION_BLOCK FB_Average
VAR_INPUT
	rValue : 			REAL;			(*Uśredniana wartość*)
	tInterval : 		TIME;			(*Co jaki czas ma byc robiony wpis*)
END_VAR
VAR_OUTPUT
	rAverage: 			REAL; 			(*Wartość średnia*)
END_VAR
VAR CONSTANT
	MAX_INDEX: 			USINT 	:= 20 ;	(*Ilość wpisów do uśredniania*)
END_VAR
VAR
	aData: 				ARRAY[0..MAX_INDEX] OF REAL;
	nIndex:		 		USINT;			(*Ostatni wpis, czyli przyjmuje wartosci od 0 do MAX_INDEX - 1*)
	i:					USINT;			(*Iterator*)
	ttimer: 			TON;
	suma: 				REAL;
END_VAR

ttimer(IN:= NOT ttimer.Q, PT:= tInterval, Q=> , ET=> );

IF nIndex = 0 THEN	(*Na poczatku wypelniamy pierwsza komorke w tablicy*)
	nIndex := 1;
	aData[0] := rValue;
END_IF

IF ttimer.Q THEN
	suma := 0;
	FOR i := 1 TO nIndex DO
		aData[i - 1] := aData[i];
		suma := suma + aData[i];
	END_FOR
	IF	nIndex < (MAX_INDEX) THEN
		nIndex := nIndex + 1;
	END_IF
	aData[nIndex] := rValue;
END_IF

rAverage := suma/nIndex;

END_FUNCTION_BLOCK

// ---- POUs/Various/FB_CERHOST.TcPOU
(****************************************************************************************************)
(*							Beckhoff Automation Poland												*)
(*								FB_CERHOST v1.1														*)
(*						v1.1 - Optymalizacja kodu													*)
(*									14.07.2015														*)
(*					Blok funkcyjny aktywacji i dezatywacji apkiacji CERHOST							*)
(*						     w sterownika z system Windows CE										*)
(*	!!!!!!!!!!!!!!!!!!!!!!!!!!!!!!!!!!!!!!!!!!!!!!!!!!!!!!!!!!!!!!!!!!!!!!!!!!!!!!!!!!!!!!!!!!!!!!!!*)
(*      	UWAGA PO WYKONANIU BLOKU STEROWNIK WYKONUJE AUTOMATYCZNY RESTART						*)
(* 							Wymaga biblioteki TcUtilities.lib 										*)
(*__________________________________________________________________________________________________*)

FUNCTION_BLOCK FB_CERHOST
VAR_INPUT
	bEnableCERHOST		: BOOL;							(*  CERHOST will be enabled with a positive edge at the bEnableCERHOST.  *)
	bDisableCERHOST		: BOOL;							(*  CERHOST will be disabled with a positive edge at the bDisableCERHOST.  *)
END_VAR
VAR_OUTPUT
	bBusy				: BOOL;							(*  When the function block is activated this output is set. It remains set until and acknowledgement is received.  *)
	bError				: BOOL;							(*  If an ADS error should occur during the execution of the command, then this output is set, after the bBusy output has been reset.  *)
	nErrId				: UDINT;							(*  When the bError output is set, this variable supplies the ADS error or the command-specific error code (table).  *)
END_VAR
VAR
	fbRegSetValue		: FB_RegSetValue;				(*  This function block is used to write a data in the system registry.  *)
	sEnableData			: STRING(12) := 'CeRDisp.exe';	(*  This value come from CeRemoteDisplay_Enable.reg file.  *)
	sDisableData		: STRING(12) := '_CeRDisp.exe';	(*  This value come from CeRemoteDisplay_Disable.reg file.  *)
	tTimeOut			: TIME :=DEFAULT_ADS_TIMEOUT;
	ntReboot			: NT_Reboot;					(*  This function block is used to reboot system. *)
	rtEnableRising		: R_TRIG;						(*  Positive edge detection at the bEnableCERHOST. *)
	rtDisableRising		: R_TRIG;						(*  Positive edge detection at the bDisableCERHOST. *)
	ftBusyFalling		: F_TRIG;						(*  Negative edge detection at the fbRegSetValue.bBusy. *)
END_VAR

rtEnableRising( CLK := bEnableCERHOST );
rtDisableRising( CLK := bDisableCERHOST );

IF rtEnableRising.Q THEN
	fbRegSetValue.cbData		:= INT_TO_UDINT(LEN(sEnableData) + 1);
	fbRegSetValue.pData			:= ADR(sEnableData);
ELSIF rtDisableRising.Q THEN
	fbRegSetValue.cbData		:= INT_TO_UDINT(LEN(sDisableData) + 1);
	fbRegSetValue.pData			:= ADR(sDisableData);
END_IF

fbRegSetValue(
	sNetId		:=''	,
	sSubKey	:=	'init',
	sValName	:=	'Launch90',
	eValType	:=	REG_SZ,
	bExecute	:=	rtEnableRising.Q OR rtDisableRising.Q,
	tTimeOut	:=	tTimeOut,
	bBusy		=>	bBusy,
	bError		=>	bError,
	nErrId		=>	nErrId );

(* Reboot system only when writing to the registry has been successful. *)
ftBusyFalling (CLK := fbRegSetValue.bBusy );
ntReboot(
	NETID	:='' ,
	START	:= ftBusyFalling.Q AND NOT fbRegSetValue.bError,
	TMOUT	:= tTimeOut );

END_FUNCTION_BLOCK

// ---- POUs/Various/FB_DiskFreeSpace.TcPOU
(************************************************************************************************)
(*							Beckhoff Automation Poland											*)
(*								FB_DiskFreeSpace  v1.0											*)
(*									08.12.2014													*)
(*	Blok funkcyjny realizuje odczyt dostępnego wolnego miejsca na karcie sterownika.			*)
(*	Odczytywana wartość jest wyrażona w MegaBytes												*)
(*	Wymaga biblioteki TcMDP.lib 																*)
(*______________________________________________________________________________________________*)

FUNCTION_BLOCK FB_DiskFreeSpace
VAR_INPUT
    sAmsNetId            		: T_AmsNetId;                  (* keep empty '' for the local device *)
	bReadRequest				: BOOL	:= TRUE;
END_VAR
VAR_OUTPUT
	lrDriveFreeSpace           :LREAL;
END_VAR
VAR
	fbScanMDP					: FB_MDP_ScanModules;
	fbReadMDP					: FB_MDP_Read;
	iState						: UINT	:= 0;
	iDriveFreeSpace				:ARRAY [1..2] OF DWORD;
END_VAR

CASE iState  OF
0: (* Idle *)
	IF bReadRequest THEN
		bReadRequest	:= FALSE;
		iState			:= 1;
	END_IF
1: (* Scan for module *)
	fbScanMDP(
		bExecute:= TRUE,
		nModuleType:= eMDP_ModT_DiskManagement,
		sAmsNetId:= sAmsNetId);
	iState	:= 2;
2: (* Get received dynamic module id *)
	fbScanMDP(
		bExecute:= FALSE,
		nModuleType:= eMDP_ModT_DiskManagement);

	IF NOT fbScanMDP.bBusy THEN
		IF NOT fbScanMDP.bError THEN
			iState	:= 3;
		ELSE
			iState	:= 0;
		END_IF
	END_IF
3: (* Request MDP Element *)
	fbReadMDP.stMDP_DynAddr.nArea		:= INT_TO_BYTE(eMDP_Area_ConfigArea);
	fbReadMDP.stMDP_DynAddr.nModuleId	:= fbScanMDP.nDynModuleId;
	fbReadMDP.stMDP_DynAddr.nTableId	:= 6;
	fbReadMDP.stMDP_DynAddr.nSubIdx	:= 1;

	fbReadMDP(
		bExecute:= TRUE,
		pDstBuf:= ADR(iDriveFreeSpace),
		cbDstBufLen:= SIZEOF(iDriveFreeSpace),
		sAmsNetId:= sAmsNetId );
	iState	:= 4;
4: (* Get received Information *)
	fbReadMDP(
		bExecute:= FALSE,
		stMDP_DynAddr:= ,
		pDstBuf:= ADR(iDriveFreeSpace),
		cbDstBufLen:= SIZEOF(iDriveFreeSpace));

	IF NOT fbReadMDP.bBusy THEN
		iState	:= 0;
	END_IF
END_CASE


lrDriveFreeSpace :=DWORD_TO_LREAL(  iDriveFreeSpace[2] )* 4294967296.0 + DWORD_TO_LREAL(iDriveFreeSpace[1]) ; (*Bytes*)
lrDriveFreeSpace := lrDriveFreeSpace / 1024;	(* kB*)
lrDriveFreeSpace := lrDriveFreeSpace / 1024;  (*MB*)

END_FUNCTION_BLOCK

// ---- POUs/Various/FB_FilterEx.TcPOU
//==================================================================================================
//							Beckhoff Automation Poland
//									23.11.2016
//			Bloczek do filtru inercyjnego do wygladzania przebiegow,					
//					czas próbkowania wyliczany wewnętrznie
//  v1.1	|| TC v 3.1.4020.28		|| - poprawienie inicjalizacji, notacja wegierska
// 	v1.0	|| TC v 3.1.4020.0		|| - pierwsza wersja
//==================================================================================================
FUNCTION_BLOCK FB_FilterEx
VAR_INPUT
	rIn										: REAL;					// Sygnal wejsciowy
	tTimeConstant							: TIME;					// Stala czasowa T gdy rOut = 0,63 * rIn 
END_VAR
VAR_OUTPUT
	rOut									: REAL;					// Przefiltrowany sygnal wyjsciowy, 
END_VAR
VAR
	rLastOut								: REAL;					// Wartosc wyjscia w poprzednim cyklu
	rCycleTime								: REAL; 				// [ms]
	rTimeConst								: REAL;					// [ms]
	tX										: TIME;					// Aktualny czas
	tY 										: TIME;					// Zmienna pomocnicza, poprzedni czas
	tCycleTime								: TIME;					// Wyliczony czas cyklu
	bFirstCycle								: BOOL := TRUE;			// Flaga pierwszego cyklu - nie mamy jeszce wyliczonego prawidlowo czasu cylu 
																	// - potrzebujemy dwoch cylki do odjecia czasu
END_VAR

// Obliczenie czasu cyklu do inkrementu
tX 					:= TIME();
IF NOT bFirstCycle THEN
	tCycleTime 		:= tX - tY;
END_IF
tY 					:= tX;
// Przeliczenie czasu na typ REAL
rCycleTime 			:= TIME_TO_REAL(tCycleTime);
rTimeConst 			:= TIME_TO_REAL(tTimeConstant);
// Wyliczenie wyjscia tylko jesli stala czasowa wieksza od 1 ms i zakonczylismy inicjalizacje
IF NOT bFirstCycle AND rTimeConst > 0.001 THEN
	rOut 			:= rLastOut + (rIn - rLastOut) * rCycleTime/rTimeConst;
	rLastOut 		:= rOut;
END_IF
// Zerowanie flagu pierwszego cyklu
bFirstCycle 		:= FALSE;

END_FUNCTION_BLOCK

// ---- POUs/Various/FB_Generator.TcPOU
(************************************************************************************************)
(*							Beckhoff Automation Poland											*)
(*								FB_Generator	 v1.0											*)
(*									26.06.2008													*)
(*					Blok funkcyjny posiadający funkje generatora. Możemy wybierać typ			*)
(*					przebiegu, to czy okres będzie określony czasem czy ilością cykli programu.	*)
(*					Generator posiada również wejście RESET, które gdy przyjmuję wartość		*)
(*					powoduje pojawienie się na wyjściu wartości 0. 								*)
(*______________________________________________________________________________________________*)

FUNCTION_BLOCK FB_Generator
VAR_INPUT
	MODE:GEN_MODE;		(* Typ przebiegu :
								TRIANGLE lub 0			Przebieg trójkątny od wartości AMPL do - AMPL
								TRIANGLE_POS lub 1		Przebieg trójkątny od wartości AMPL do 0
								SAWTOOTH_RISE lub 2	Przebieg piłokształtny rosnący od wartości -AMPL do AMPL
								SAWTOOTH_FALL lub 3	Przebieg piłokształtny opadający od wartości AMPL do -AMPL
								RECTANGLE lub 4		Przebieg prostokątny AMPL i - AMPL 
								SINUS lub 5				Przebieg sinusoidalny
								COSINUS lub 6			Przebieg cosinusoidalny *)
	BASE:BOOL;			(* Okleślenie okresu : FALSE-Liczba cykli programu ; TRUE-Czas *)
	PERIOD:TIME;		(* Okres, jeżeli BASE=TRUE *)
	CYCLES:INT;			(* Cykle programu na okres, jeżeli BASE=FALSE *)
	AMPLITUDE:INT;		(* Amplituda *)
	RESET:BOOL;			(* Reset *)
END_VAR
VAR_OUTPUT
	OUT:INT;
END_VAR
VAR
	CET,PER:DWORD;
	COUNTER:INT;
	CLOCK:TON;
END_VAR

IF RESET THEN
	COUNTER:=0;
	OUT:=0;
	CLOCK(IN:=FALSE);
ELSE
	IF BASE=FALSE THEN		(* Periodizität bzgl. Aufrufe *)
		COUNTER:=(COUNTER+1)MOD CYCLES;
		CASE MODE OF
		0:	(* Dreiecksfunktion von -AMPL bis AMPL.*)
			OUT:=(CYCLES-2*ABS(CYCLES-2*COUNTER))*AMPLITUDE/CYCLES;
		1:	(* Dreiecksfunktion von 0 bis AMPL.*)
			OUT:=(CYCLES-ABS(CYCLES-2*COUNTER))*AMPLITUDE/CYCLES;
		2:	(* Sägezahn steigend *)
			OUT:=(2*COUNTER-CYCLES)*AMPLITUDE/CYCLES;
		3:	(* Sägezahn fallend *)
			OUT:=(CYCLES-2*COUNTER)*AMPLITUDE/CYCLES;
		4:	(* Rechteck AMPL./-AMPL. *)
			IF 2*COUNTER>CYCLES THEN
				OUT:=-AMPLITUDE;
			ELSE
				OUT:=AMPLITUDE;
			END_IF
		5:	(* Sinusfunktion *)
			OUT:=REAL_TO_INT(SIN(6.283167*COUNTER/CYCLES)*AMPLITUDE);
		6:	(* Cosinusfunktion *)
			OUT:=REAL_TO_INT(COS(6.283167*COUNTER/CYCLES)*AMPLITUDE);
		END_CASE;
	ELSE												(* Periodizität bzgl. Zeit *)
		CLOCK();										(* Timer abfragen *)
		IF CLOCK.PT<>PERIOD+PERIOD THEN	(* Initialisierung *)
			CLOCK.PT:=PERIOD+PERIOD;		(* Setze Timer auf zwei PERIODn *)
			CLOCK(IN:=TRUE);
		ELSE
			CET:=TIME_TO_DWORD(CLOCK.ET);
			PER:=TIME_TO_DWORD(PERIOD);
			IF CET>=PER THEN	(* Neuinitialisierung des Timers*)
				CLOCK(IN:=FALSE);
				CLOCK(IN:=TRUE);
				CET:=CET MOD PER;
			END_IF
			CASE MODE OF
			0:	(* Dreiecksfunktion -AMPL bis AMPL.*)
				OUT:=(1-2*ABS(1-2*DWORD_TO_INT(CET/PER))*AMPLITUDE);
			1:	(* Dreiecksfunktion 0 bis AMPL.*)
				OUT:=(1-ABS(1-2*DWORD_TO_INT(CET/PER))*AMPLITUDE);
			2:	(* Sägezahn steigend *)
				OUT:=((2*DWORD_TO_INT(CET/PER)-1)*AMPLITUDE);
			3:	(* Sägezahn fallend *)
				OUT:=((1-2*DWORD_TO_INT(CET/PER))*AMPLITUDE);
			4:	(* Rechteck AMPL./-AMPL. *)
				IF CET*2<PER THEN
					OUT:=-AMPLITUDE;
				ELSE
					OUT:=AMPLITUDE;
				END_IF
			5:	(* Sinusfunktion *)
				OUT:=REAL_TO_INT(SIN(6.283167*DWORD_TO_REAL(CET/PER))*AMPLITUDE);
			6:	(* Cosinusfunktion *)
				OUT:=REAL_TO_INT(COS(6.283167*DWORD_TO_REAL(CET/PER))*AMPLITUDE);
			END_CASE;
		END_IF
	END_IF;
END_IF;

END_FUNCTION_BLOCK

// ---- POUs/Various/FB_Hysteresis.TcPOU
(************************************************************************************************)
(*							Beckhoff Automation Poland											*)
(*								FB_Hysteresis v1.0												*)
(*									9.02.2011													*)
(*				Blok funkcyjny histerezy. Zaczyna pracę z wyjsciem ustawionym na FALSE			*)
(*					Histereza w obrzasze rSetValue - rH1<	...	<rSetValue + rH2				*)
(*			Dla warości wejściowej rActualValue < rSetValue - rH1przyjmuje wartość FALSE		*)
(*			Dla warości wejściowej rActualValue > rSetValue + rH2przyjmuje wartość TRUE			*)
(*______________________________________________________________________________________________*)
FUNCTION_BLOCK FB_Hysteresis
VAR_INPUT
	bEnable: 		BOOL:=TRUE;
	rActualValue: 	REAL;
	rSetValue: 		REAL;
	rH1: 			REAL;
	rH2: 			REAL;
END_VAR
VAR_OUTPUT
	bOut: 			BOOL;
END_VAR

IF bEnable THEN
	IF rActualValue <= rSetValue - rH1 THEN bOut := FALSE; END_IF
	IF rActualValue >= rSetValue + rH2 THEN bOut := TRUE; END_IF
ELSE
	bOut := FALSE;
END_IF

END_FUNCTION_BLOCK

// ---- POUs/Various/FB_Persistent.TcPOU
FUNCTION_BLOCK FB_Persistent

(********************************************************************************************************)
(*								Beckhoff Automation Poland												*)
(* 									FB_Persistent 	v1.5												*)
(* 										20.08.2014														*)
(* 							v1.5 - zmiana minimalnego interwalu zapisu									*)
(* 					Blok funkcyjny zapisujący zmienne typu persistent na karcie CF						*)
(* 						Możliwy zapis na żądanie lub z określoną częstotliwością.  						*)
(* 				Pozostawienie wejscia tInterval bez zmiennej wyłacza funkcję zapisu cyklicznego			*)
(* 							Minimalny czas między zapisem cyklicznym 30s								*)
(* 				Konieczne jest dodanie biblioteki TcUtilities.lib, TcSystem.lib oraz TcBase.lib			*)
(*			 UWAGA: Blok przygotowany dla RunTime 1 port 801 - typowa konfiguracja 						*)
(*______________________________________________________________________________________________________*)

VAR_INPUT
	bWrite					: BOOL;						(*Zapis na rozkaz *)
	tInterval				: TIME:=T#71582M47S295MS;	(*Czestotliwosc zapisu na karte CF*)
END_VAR
VAR_OUTPUT
	bBusy					: BOOL;
	bErr					: BOOL;
	udErrID					: UDINT;
END_VAR
VAR
	fbWritePersistentData	: FB_WritePersistentData; 	(* Blok zapisu *)
	t1						: TON;						(* Timer zapisu *)
	_GETCURTASKINDEX		: GETCURTASKINDEX;			(* Informacja o Tasku *)
	BIndex					: BYTE;						(* Nr tasku *)
END_VAR

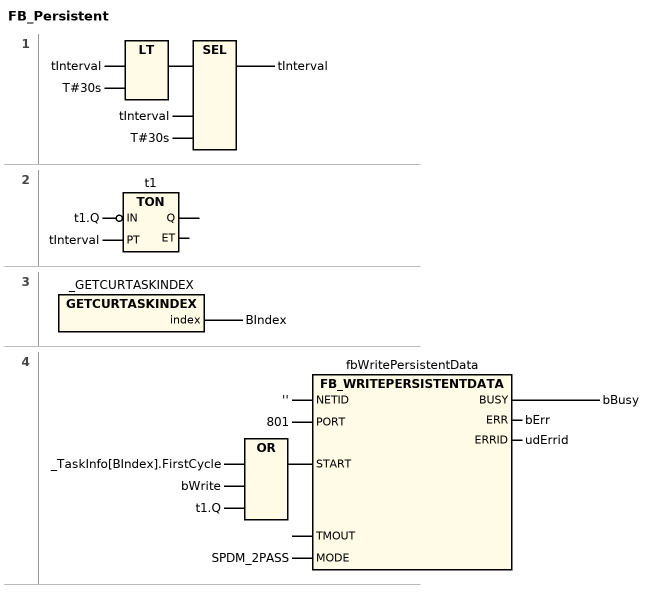
// NETWORK 1
tInterval := SEL(tInterval < T#30s, tInterval, T#30s);

// NETWORK 2
t1(IN := NOT t1.Q, PT := tInterval); // TON

// NETWORK 3
_GETCURTASKINDEX(); // GETCURTASKINDEX
BIndex := _GETCURTASKINDEX.index;

// NETWORK 4
fbWritePersistentData(
    NETID := '',
    PORT := 801,
    START := _TaskInfo[BIndex].FirstCycle OR bWrite OR t1.Q,
    MODE := SPDM_2PASS,
    ERR => bErr,
    ERRID => udErrid); // FB_WRITEPERSISTENTDATA
bBusy := fbWritePersistentData.BUSY;

END_FUNCTION_BLOCK

// ---- POUs/Various/FB_PIDBasic.TcPOU
//==================================================================================================
//					Beckhoff Automation Poland
//							18.11.2016
//		Blok funkcyjny regulatora PID w wersji podstawowej
// 	v1.0 	|| TC v 3.1.4020.28 	|| - pierwsza wersja
//==================================================================================================
FUNCTION_BLOCK FB_PIDBasic
VAR_INPUT
	bEnable				: BOOL; 			// Pozdolenie na dzialanie, FALSE - resetuje zawartosc
	bInvertDirection	: BOOL; 			// TRUE: Heating
	lrSetpointValue		: LREAL; 			// Wartosc zadana
	lrActualValue		: LREAL; 			// Wartosc aktualna
	bReset				: BOOL;				// Restart bloku
	bFreeze				: BOOL;				// Zatrzasniecie wyjscia
	bManual				: BOOL;				// Tryb reczny
	lrManual			: LREAL;			// Wartosc dla trybu recznego
	lrYMin				: LREAL;			// Ograniczenie dolne wyjscia
	lrYMax				: LREAL;			// Ograniczenie gorne wyjscia
	lrKp				: LREAL;			// Wzmocnieie proporcjonalne
	tTn					: TIME; 			// Stala czasowa ocji calkujacej
	tTv					: TIME; 			// Stala czasowa akcji rozniczkujacej
	tTd					: TIME; 			// Stala czasowa akcji rozniczkujacej
	lrTaskCycleTime		: LREAL; 			// Czas tasku w ms
	lrCycleTime			: LREAL; 			// Interwal wywolania obliczen w ms - powinna to byc wielokrotnosc cyklu
END_VAR
VAR_OUTPUT
	lrY					: LREAL; 			// Wyjscie
	lrE					: LREAL; 			// Odchylka regulacji
	bActive				: BOOL; 			// Regulator dziala
	bARWactive			: BOOL; 			// Ochrona calkowania
	bMinLimit			: BOOL; 			// Limit gorny
	bMaxLimit			: BOOL; 			// Limit dolny
	bError				: BOOL; 			// Blad parametru
END_VAR
VAR
	bExecutionCycle		: BOOL;
	bInit				: BOOL;
	bIPartEnabled		: BOOL;
	bDPartEnabled		: BOOL;
	bCtrlDisabled		: BOOL;
	uiCycle				: UINT;
	uiCycleCall			: UINT;
	lrTn				: LREAL;
	lrTv				: LREAL;
	lrTd				: LREAL;
	lre_1				: LREAL;
	lrYP				: LREAL;
	lrYI				: LREAL;
	lrYI_1				: LREAL;
	lrYD				: LREAL;
	lrYD_1				: LREAL;
	lrY_1				: LREAL;
	lrdI				: LREAL;
	lrdD				: LREAL;
	lrcD				: LREAL;
	lrY_Test			: LREAL;
END_VAR

	bError		:= FALSE;
	IF lrTaskCycleTime < 0.001 THEN bError := TRUE; END_IF
	IF lrCycleTime < lrTaskCycleTime THEN bError	:= TRUE; END_IF
	IF lrYMin>=lrYMax THEN bError := TRUE; END_IF
	IF (lrKp<0.0) THEN bError := TRUE; END_IF
	IF bError THEN RETURN; 	END_IF


IF NOT bEnable OR NOT bInit	THEN
	lrY				:= 0.0;
	lrE				:= 0.0;
	lrE_1			:= 0.0;
	lrYP			:= 0.0;
	lrYI			:= 0.0;
	lrYI_1			:= 0.0;
	lrYD			:= 0.0;
	lrYD_1			:= 0.0;
	lrY_Test		:= 0.0;
	bARWactive		:= FALSE;
	bActive			:= FALSE;
	uiCycle			:= 1;
	bInit			:= TRUE;
	IF NOT bEnable THEN RETURN; END_IF
END_IF
(* Flagi i limity *)
bActive	:= TRUE;
bIPartEnabled := tTn > t#0ms; (*Czy jest czlon I?*)
bDPartEnabled := tTv > t#0ms; (*Czy jest czlon D?*)
lrManual := LIMIT(lrYMin, lrManual, lrYMax);	(* Manual musi byc w limitach *)

(*Konwersja czasow*)
lrTn	:= TIME_TO_LREAL(tTn);
lrTv	:= TIME_TO_LREAL(tTv);
lrTd	:= TIME_TO_LREAL(tTd);

(*Wyliczenie co ile cykli jest obliczenie wyjscia*)
uiCycleCall := LREAL_TO_INT(lrCycleTime/lrTaskCycleTime);

(*Obliczenie wspolczynnikow czlonow I i D*)
IF tTn>t#0ms THEN
	lrdI :=	(lrCycleTime/2.0)/lrTn;
END_IF
lrdD :=	lrTv/(lrTd+(lrCycleTime/2.0));
lrcD :=	(lrTd-(lrCycleTime/2.0))/(lrTd+(lrCycleTime/2.0));

(* Obliczenia w kazdym pierwszym cyklu *)
bExecutionCycle := uiCycle = 1;
(* Iterowanie cykli obliczeniowych, obliczenia tylko w cyklu 1, ale to dalej *)
uiCycle:=uiCycle+1;
IF (uiCycle > uiCycleCall) THEN uiCycle:=1; END_IF;

(* Jak obliczenia nie teraz, to wroc *)
IF NOT bExecutionCycle	THEN
	RETURN;
END_IF

(**********************************Regulator PID**********************************)
(*Przepisanie wartosci z poprzedniego cyklu*)
lrE_1	:= lrE;
lrYI_1	:= lrYI;
lrYD_1	:= lrYD;
lrY_1	:= lrY;

(* Kierunek - wprost czy odwrocony*)
lrE := SEL(bInvertDirection, lrActualValue-lrSetpointValue, -(lrActualValue-lrSetpointValue)); (* bInvertDirection = TRUE --> grzanie *)

(*Blokada regulacji gdy mamy minimum i odchylke mniejsza/rowna 0, lub gdy mamy maks i odchylke wieksza/rowna 0*)
bCtrlDisabled:=(bMinLimit AND (lrE <= 0.0)) OR	(bMaxLimit AND (lrE >= 0.0));

(* Jak manual to resetujemy blokadę*)
IF	bManual	THEN bCtrlDisabled:=FALSE; END_IF

bARWactive:=bCtrlDisabled;

(*+++++++++++++++++++++++++++++*)
(*P-I-D-Obliczenia*)
IF NOT bCtrlDisabled	THEN
	(*Czlon: P*);
	lrYP:=lrKp*lrE;
	(*Czlon: I*)
	IF bIPartEnabled THEN
		lrYI:=lrdI*(lrE+lrE_1)+lrYI_1;
	ELSE
		lrYI		:=0;
		lrYI_1	:=0;
	END_IF
	(*Czlon: D*)
	IF bDPartEnabled 	THEN
		IF (lrTd <= lrCycleTime) THEN
			lrYD:= (lrTv/lrCycleTime) * (lrE-lrE_1);
		ELSE
			lrYD:= (lrcD*lrYD_1)+(lrdD*(lrE-lrE_1));
		END_IF
	ELSE
		lrYD		:=0;
		lrYD_1	:=0;
	END_IF
END_IF

(*Sprawdzenie czy nie przekroczymy limitów - w razie potrzeby obcinamy I i D zeby wyrownac do limitu*)
lrY_Test:=lrYP+lrYI+lrYD;
IF NOT bCtrlDisabled THEN
	IF lrY_Test<lrYMin	THEN
		IF		bIPartEnabled THEN
					lrYI:=lrYMin-lrYP-lrYD;
		ELSIF	bDPartEnabled THEN
					lrYD:=lrYMin-lrYP;
		END_IF
	END_IF
	IF lrY_Test>lrYMax THEN
		IF		bIPartEnabled THEN
					lrYI:=lrYMax-lrYP-lrYD;
		ELSIF	bDPartEnabled THEN
					lrYD:=lrYMax-lrYP;
		END_IF
	END_IF
END_IF

(*Jak odciecie sterowania - wyliczenie nowych czlonow I i D*)
IF bCtrlDisabled	THEN
	IF bMinLimit	THEN
		IF		bIPartEnabled THEN
					lrYI:=lrYMin-lrYP-lrYD;
		ELSIF	bDPartEnabled THEN
					lrYD:=lrYMin-lrYP;
		END_IF
	END_IF

	IF bMaxLimit	THEN
		IF		bIPartEnabled THEN
					lrYI:=lrYMax-lrYP-lrYD;
		ELSIF	bDPartEnabled THEN
					lrYD:=lrYMax-lrYP;
		END_IF
	END_IF
END_IF

(*Wyliczenie wyjscia po limitach*)
lrY_Test:=lrYP+lrYI+lrYD;

(*Tryb reczny wyliczenie - wyliczenie nowych czlonow I i D*)
IF bManual	THEN
	IF		bIPartEnabled THEN
				lrYI:=lrManual-lrYP-lrYD;
	ELSIF	bDPartEnabled THEN
				lrYD:=lrManual-lrYP;
	END_IF
END_IF

(*+++++++++++++++++++++++++++++++++++++++++++++++++*)
(*Obliczenie wyjscia*)
lrY:=lrYP+lrYI+lrYD;

(* Freeze - zatrzasniecie wyjscia*)
IF bFreeze THEN
	lrYI			:= lrYI_1;
	lrYD			:= lrYD_1;
	lrY				:= lrY_1;
END_IF

(*Ograniczenie limitów*)
bMaxLimit	:= lrY>=lrYMax;
bMinLimit	:= lrY<=lrYMin;
lrY := LIMIT(lrYMin, lrY, lrYMax);

IF bReset THEN
	A_Reset();
END_IF

ACTION A_Reset:
	bExecutionCycle		:=FALSE;
	bInit				:=FALSE;
	bIPartEnabled		:=FALSE;
	bDPartEnabled		:=FALSE;
	bCtrlDisabled		:=FALSE;
	uiCycle				:=0;
	uiCycleCall			:=0;
	lrTn				:=0;
	lrTv				:=0;
	lrTd				:=0;
	lre_1				:=0;
	lrYP				:=0;
	lrYI				:=0;
	lrYI_1				:=0;
	lrYD				:=0;
	lrYD_1				:=0;
	lrY_1				:=0;
	lrdI				:=0;
	lrdD				:=0;
	lrcD				:=0;
	lrY_Test			:=0;
	lrY					:=0; (* Wyjscie  *)
	lrE					:=0; (* Odchylka regulacji *)
	bActive				:=FALSE; (* Regulator dziala *)
	bARWactive			:=FALSE; (* Ochrona calkowania *)
	bMinLimit			:=FALSE; (* Limit gorny *)
	bMaxLimit			:=FALSE; (* Limit dolny *)
	bError				:=FALSE; (* Blad parametru *)
END_ACTION

END_FUNCTION_BLOCK

// ---- POUs/Various/FB_Ramp.TcPOU
(****************************************************************************************)
(*							Beckhoff Automation Poland									*)
(*								FB_Ramp v1.0											*)
(*									31.09.2011											*)
(*							Blok rampy, narastanie liniowe								*)
(*______________________________________________________________________________________*)
FUNCTION_BLOCK FB_Ramp
VAR_INPUT
	rIn:			REAL; 			(* Aktualna wartość regulowana *)
	tTime:			TIME;			(* Czas co jaki dodajemy gradient wartości *)
	rMaxUp:			REAL;			(* Maksymalna wartość o jaką jednorazowo możemy zwiększyć warość wyjścia *)
	rMaxDown:		REAL;			(* Maksymalna wartość o jaką jednorazowo możemy zmniejszyć warość wyjścia *)
END_VAR
VAR_OUTPUT
	rOut:			REAL;			(* Wartość wyjściowa *)
END_VAR
VAR
	clock:			TP;
	lastOut:	 	REAL;
	stan: 			BOOL;
	oldstan: 		BOOL;
END_VAR

CLOCK();
clock.PT:=tTime;
IF CLOCK.Q=FALSE THEN
	CLOCK(IN:=FALSE);
	stan := NOT stan;
	CLOCK(IN:=TRUE);
END_IF
IF(oldstan <> stan) THEN
	IF(rIn>=lastout + rMaxUp) THEN rOut := lastout + rMaxUp; END_IF
	IF (rIn<= lastout - rMaxDown) THEN rOut := lastout - rMaxDown;END_IF
	IF(rIn<lastout + rMaxUp AND rIn > lastout - rMaxDown) THEN rOut:= rIn;END_IF
END_IF
lastout := rOut;
oldstan:=stan;

END_FUNCTION_BLOCK

// ---- POUs/Various/FB_ReadRegister.TcPOU
(************************************************************************************************)
(*							Beckhoff Automation Poland											*)
(*								FB_ReadRegister	 v1.0											*)
(*									9.9.2009													*)
(*			Blok funkcyjny odczytujacy wartosc z rejestru modułu analogowego KLxxxx				*)
(*				Szczegolowe informacje dotyczace komunikacji z rejestrami						*)
(*				i wartosci w nich przechowywanych znajduja sie w dokumentacji modulu			*)
(*				W programie może być jednocześnie wywołany 1 blok dla 1 kanalu 					*)
(*______________________________________________________________________________________________*)
FUNCTION_BLOCK FB_ReadRegister
VAR_INPUT
	bRead: 		BOOL;		(*Rozkaz odczytu*)
	iRegNo:		INT;		(*Numer odczytywanego rejestru*)
	State: 		BYTE;		(*Nalezy zlinkowac do State przy konkretnym kanale w module KLxxxx*)
	DataIn: 	INT;		(*Nalezy zlinkowac do Data_In przy konkretnym kanale w module KLxxxx*)
END_VAR
VAR_OUTPUT
	bBusy:		BOOL; 		(*Blok wykonuje akcje*)
	bError:		BOOL;		(*Wystapil blad*)
	Value: 		INT;		(*Odczytana wartosc*)
	Ctrl: 		BYTE;		(*Nalezy zlinkowac do Ctrl przy konkretnym kanale w module KLxxxx*)
END_VAR
VAR
	Step: 		INT;		(*Krok instrukcji CASE*)
	Temp: 		BYTE;		(*Zapamietanie wartosci CTRL przez odczytem*)
	rtRead:		R_TRIG;		(*Zlapanie rozkazu odczytu*)
	Timeout:	TON;		(*Wykrycie bledu*)
END_VAR

(*Sprawdzanie czy nie uplynal czas*)
	Timeout(IN:=Step<>0 , PT:= T#200ms, Q=> bError);
	IF bError THEN Step := 99; END_IF

(*Wykrycie sygnalu do odczytu*)
	rtRead(CLK:= bRead, Q=> );

(*Odczyt*)
	CASE Step OF
	0:
		(*Mierzymy chyba ze otrzymamy sygnal startu*)
		IF rtRead.Q THEN
			bBusy := TRUE;
			Step := Step+10;
		END_IF
	10:
		Temp := Ctrl;(*Zapamietanie controla sprzed odczytu*)
		Ctrl :=INT_TO_BYTE(128+iRegNo); (*1|0|Reg_No*)
		Step := Step+10;
	20:
		IF State = Ctrl THEN
			Value := DataIn;
			Ctrl := Temp;
			bBusy := FALSE;
			Step := 0;
		END_IF
	99:	(*Gdy blad*)
		Ctrl := Temp;
		bBusy := FALSE;
		Step := 0;
	END_CASE

END_FUNCTION_BLOCK

// ---- POUs/Various/FB_RecMove.TcPOU
(****************************************************************************************************)
(*							Beckhoff Automation Poland												*)
(*								FB_RecMove	 v1.0													*)
(*									29.12.2008														*)
(*		Blok funkcyjny obliczający polozenie punktu w kartezjanskim ukladzie wspolrzednych			*)
(*							po obrocie o ustaony kat												*)
(*		Wartosciami wejsciowymi jest polozenie srodka okregu, punktu startowego i katu obrotu		*)
(*__________________________________________________________________________________________________*)
FUNCTION_BLOCK FB_RecMove
VAR_INPUT
(*Srodek okregu*)
	Xs: 			REAL:=5;
	Ys:				REAL:=0;
(*Punkt poczatkowy*)
	X0: 			REAL:=0;
	Y0:				REAL:=0;
(*Kat przesuniecia*)
	alfa:			REAL:=90;
END_VAR
VAR_OUTPUT
(*Punkt koncowy*)
	X1: 			REAL;
	Y1:				REAL;
END_VAR

X1 := LREAL_TO_REAL((X0-Xs)*COS(alfa*PI/180)+Xs-(Y0-Ys)*SIN(alfa*PI/180));
Y1 := LREAL_TO_REAL((X0-Xs)*SIN(alfa*PI/180)+(Y0-Ys)*COS(alfa*PI/180)+Ys);

END_FUNCTION_BLOCK

// ---- POUs/Various/FB_SetIPAddress.TcPOU
(************************************************************************************************************************)
(*							Beckhoff Automation Poland								*)
(*								FB_SetIPAddress	 v1.0									*)
(*							v1.0 - implementacja										*)
(*									02.11.2015										*)
(*							Blok zmieniający adres IP									*)
(*	Działa na: CP6606-0020															*)
(*_______________________________________________________________________________*)
FUNCTION_BLOCK  FB_SetIPAddress
VAR_INPUT
	bSetIP				:	BOOL;
	bDHCP				:	BOOL;
	sMachineIP			: 	STRING(15);	(*192.168.1.14*)
	sMachineMask		:	STRING(15);	(*255.255.255.0*)
	sMachineGateway 	: 	STRING(15);	(*192.168.1.1*)
END_VAR
VAR_OUTPUT
	bBusy				:	BOOL;
	bError				:	BOOL;
	nErrorID				:	UDINT;
END_VAR
VAR
	iState				:	INT;
	rtSetIP				:	R_TRIG;
	fbRestart 			: 	NT_Reboot;
	fbScan				: 	FB_MDP_ScanModules;
	fbWrite				: 	FB_MDP_Write;
END_VAR

CASE iState OF
0:
	rtSetIP(CLK := bSetIP);
	IF rtSetIP.Q THEN
		iState := 10;
		bBusy := TRUE;
		bError := FALSE;
		nErrorID := 0;
	END_IF
10:
	fbScan(bExecute:=TRUE ,nModuleType:=eMDP_ModT_NIC ,iModIdx:=0);
	IF NOT fbScan.bBusy THEN
		IF NOT fbScan.bError THEN
			iState := iState + 10;
		ELSE
			iState := 999;
			nErrorID := fbScan.nErrID;
		END_IF
		fbScan( bExecute:= FALSE );
	END_IF

20: (* set DHCP *)
	fbWrite.stMDP_DynAddr.nArea     := INT_TO_BYTE(eMDP_Area_ConfigArea);
	fbWrite.stMDP_DynAddr.nModuleId := fbScan.nDynModuleId;
	fbWrite.stMDP_DynAddr.nTableId  := 1;
	fbWrite.stMDP_DynAddr.nSubIdx := 4;		(* DHCP *)
	fbWrite(bExecute:= TRUE, pSrcBuf:= ADR(bDHCP),cbSrcBufLen:= SIZEOF(bDHCP));
	IF NOT fbWrite.bBusy THEN
		IF NOT fbWrite.bError THEN
			iState := iState + 10;
		ELSE
			iState := 999;
			nErrorID := fbWrite.nErrID;
		END_IF
		fbWrite( bExecute:= FALSE );
	END_IF
30:
	fbWrite.stMDP_DynAddr.nSubIdx := 2;	(* IP address *)
	fbWrite(bExecute:= TRUE, pSrcBuf:= ADR(sMachineIP),cbSrcBufLen:= INT_TO_UDINT(LEN(sMachineIP)));
	IF NOT fbWrite.bBusy THEN
		IF NOT fbWrite.bError THEN
			iState := iState + 10;
		ELSE
			iState := 999;
			nErrorID := fbWrite.nErrID;
		END_IF
		fbWrite( bExecute:= FALSE );
	END_IF
40:
	fbWrite.stMDP_DynAddr.nSubIdx := 3;	(* Mask *)
	fbWrite(bExecute:= TRUE, pSrcBuf:= ADR(sMachineMask), cbSrcBufLen:= INT_TO_UDINT(LEN(sMachineMask)));
	IF NOT fbWrite.bBusy THEN
		IF NOT fbWrite.bError THEN
			iState := iState + 10;
		ELSE
			iState := 999;
			nErrorID := fbWrite.nErrID;
		END_IF
		fbWrite( bExecute:= FALSE );
	END_IF

50:
	fbWrite.stMDP_DynAddr.nSubIdx := 5;	(* Gateway *)
	fbWrite(bExecute:= TRUE, pSrcBuf:= ADR(sMachineGateway), cbSrcBufLen:= INT_TO_UDINT(LEN(sMachineGateway)));
	IF NOT fbWrite.bBusy THEN
		IF NOT fbWrite.bError THEN
			iState := iState + 10;
		ELSE
			iState := 999;
			nErrorID := fbWrite.nErrID;
		END_IF
		fbWrite( bExecute:= FALSE );
	END_IF
60:
	fbRestart(
		NETID:= ,
		DELAY:= ,
		START:=TRUE ,
		TMOUT:= ,
		BUSY=> ,
		ERR=> ,
		ERRID=> );
	IF NOT fbRestart.BUSY THEN
		IF NOT fbRestart.ERR THEN
			iState := 0;
			bBusy := FALSE;
		ELSE
			iState := 999;
			nErrorID := fbRestart.ERRID;
		END_IF
	END_IF
999:
	iState :=0;
	bError := TRUE;
	bBusy := FALSE;
	fbWrite( bExecute:= FALSE );
	fbRestart(START:=FALSE);
	fbScan( bExecute:= FALSE );
END_CASE

END_FUNCTION_BLOCK

// ---- POUs/Various/FB_SinGenerator.TcPOU
//==================================================================================================
//					Beckhoff Automation Poland
//							02.02.2017
//		Blok funkcyjny generujacy sinusoide o zadanej amplitudzie i okresie
// 	v1.0 	|| TC v 3.1.4020.28 	|| - pierwsza wersja
//==================================================================================================
FUNCTION_BLOCK FB_SinGenerator
VAR_INPUT
	bEnable						: BOOL;							// TRUE - obliczamy wyjscie, FALSE - zerujemy wyjscie
	bReset						: BOOL;							// zeruje wartosci
	lrAmplitude					: LREAL;						// amplituda wyjscia
	tPeriod						: TIME;							// okres sinusoidy w ms
	lrOffset					: LREAL;						// offset wyjscia
	lrPeriodOffset				: LREAL;						// offset w okresie 0..T, np. 0.25 oznacza 1/4 okresu, 
																// w przypadku wartosci wiekszych od 1 brana jest tylk czesc ulamkowa
END_VAR
VAR_OUTPUT
	lrOut						: LREAL;						// wartosc wyjsciowa
END_VAR
VAR
	diTaskIndex					: DINT;							// index tasku
	lrTaskTime					: LREAL;						// czas tasku
	lrPeriod					: LREAL;						// okres sinusoidy w ms
	lrDeltaTime					: LREAL;						// przyrost czas tasku/okres, o ile na sinusoidzie przesuwamy sie w czasie znormalizowanym
	lrTime						: LREAL;						// czas od podania enable
	bFirstCycle					: BOOL := TRUE;					// flaga pierwszego cyklu
END_VAR

IF bFirstCycle OR bReset THEN
	diTaskIndex 				:= GETCURTASKINDEXEX();												// pobranie numeru tasku
	lrTaskTime 					:= UDINT_TO_LREAL(_TaskInfo[diTaskIndex].CycleTime)/10000.0;		// pobranie czasu cyklu w ms
	lrTime 						:= lrPeriodOffset;
	lrOut						:= 0.0;																// wyzerowanie wyjscia
	bFirstCycle 				:= FALSE;
END_IF
IF bEnable THEN
	lrPeriod 					:= TIME_TO_LREAL(tPeriod);											// w ms
	IF lrPeriod < 1.0 THEN 		lrPeriod := 1.0; END_IF
	lrDeltaTime					:= lrTaskTime / lrPeriod;											//
	lrOut 						:= (lrAmplitude * SIN(lrTime * 2.0 * PI)) + lrOffset;				// wyliczenie wyjscia
	lrTime						:= lrTime + lrDeltaTime;											// inkrement
ELSE
	lrOut						:= 0.0;																// wyzerowanie wyjscia
	bFirstCycle					:= TRUE;															// ustawienie flagi pierwszego cyklu
END_IF

END_FUNCTION_BLOCK

// ---- POUs/Various/FB_WriteRegister.TcPOU
(***************************************************************************************************************************)
(*							Beckhoff Automation Poland									*)
(*								FB_WriteRegister	 v1.0										*)
(*									9.9.2009												*)
(*			Blok funkcyjny zapisujacy wartosc do rejestru modułu analogowego KLxxxx				*)
(*				Szczegolowe informacje dotyczace komunikacji z rejestrami						*)
(*				i wartosci w nich przechowywanych znajduja sie w dokumentacji modulu			*)
(*				W programie może być jednocześnie wywołany 1 blok dla 1 kanalu 				*)
(*_______________________________________________________________________________________*)
FUNCTION_BLOCK FB_WriteRegister
VAR_INPUT
	bWrite: 		BOOL;	(*Rozkaz zapisu*)
	iRegNo:		INT;		(*Numer zapisywanego  rejestru*)
	Value: 		INT;		(*Wpisana wartosc*)
	State: 		BYTE;	(*Nalezy zlinkowac do State przy konkretnym kanale w module KLxxxx*)
	DataIn: 		INT;		(*Nalezy zlinkowac do Data_In przy konkretnym kanale w module KLxxxx*)
END_VAR
VAR_OUTPUT
	bBusy:		BOOL; 	(*Blok wykonuje akcje*)
	bError: 		BOOL;	(*Wystapil blad*)
	Ctrl: 			BYTE;	(*Nalezy zlinkowac do Ctrl przy konkretnym kanale w module KLxxxx*)
	DataOut: 	INT;		(*Nalezy zlinkowac do Data_Out przy konkretnym kanale w module KLxxxx*)
END_VAR
VAR
	Step: 		INT;		(*Krok instrukcji CASE*)
	Temp: 		BYTE;	(*Zapamietanie wartosci CTRL przez zapisem*)
	rtWrite:		R_TRIG;	(*Zlapanie rozkazu zapisu*)
	Timeout:		TON;	(*Wykrycie bledu*)
END_VAR

(*Sprawdzanie czy nie uplynal czas*)
	Timeout(IN:=Step<>0 , PT:= T#200ms, Q=> bError);
	IF bError THEN Step := 99; END_IF

(*Wykrycie sygnalu do odczytu*)
	rtWrite(CLK:= bWrite, Q=> );

(*Zapis*)
	CASE Step OF
	0:	(*Mierzymy chyba ze otrzymamy sygnal startu*)
		IF rtWrite.Q THEN
			bBusy := TRUE;
			Step := Step+10;
		END_IF
	10:	(*Otwarcie rejestrow do zapisu*)
		Ctrl:=2#11011111; (* otwieramy do zapisu R31*)
		DataOut:=16#1235; (* i wpisujemy 1235 hex*)
		Step:=Step+10;
	20:	(*Jezeli sa otwarte to wpisujemy*)
		IF State=2#10011111 THEN
			Ctrl :=INT_TO_BYTE(192+iRegNo); (*1|1|Reg_No*)
			DataOut :=Value;
			Step:=Step+10;
		END_IF
	30:	(*Jezeli udalo sie wpisac, to zamykamy rejestry*)
		IF State=INT_TO_BYTE(128+iRegNo) THEN
			Ctrl:=2#11011111; (* otwieramy do zapisu R31*)
			DataOut:=16#0; (* i wpisujemy 1235 hex*)
			Step:=Step+10;
		END_IF
	40:	(*Zamykamy rejestry*)
		IF State=2#10011111 THEN
			Ctrl :=Temp;
			DataOut :=0;
			bBusy := FALSE;
			Step:=0;
		END_IF
	99:	(*Gdy blad*)
		Ctrl := Temp;
		DataOut := 0;
		bBusy := FALSE;
		Step := 0;
	END_CASE

END_FUNCTION_BLOCK

// ---- POUs/Various/F_CRC_CALC.TcPOU
(************************************************************************************)
(*							Beckhoff Automation Poland								*)
(*								F_CRC_CALC v1.0										*)
(*									6.07.2015										*)
(*							Funkcja obliczajaca CRC-CCITT 							*)
(*__________________________________________________________________________________*)
FUNCTION F_CRC_CALC 	: WORD
VAR_INPUT
	wCrc_buff			: WORD;
	byInput				: BYTE;
END_VAR
VAR
	i					: BYTE;
	wX16				: WORD;
END_VAR

